// TwinCAT 3 PLC project IBF_Devices
// Title: IBF_Device
// Company: Industrial Brains B.V.
// ProjectVersion: 0.0.0.0
// ProgramVersion: 3.1.4022.4
// CompilerDefines: InclSerialCom := 'true'
// libraries:
//   IBF_Utilities, * (Industrial Brains B.V.)
//   Tc2_Math, * (Beckhoff Automation GmbH)
//   Tc2_MC2, * (Beckhoff Automation GmbH)
//   Tc2_MC2_Drive, * (Beckhoff Automation GmbH)
//   Tc2_Standard, * (Beckhoff Automation GmbH)
// project tree:
//   Actuators/Cylinder/DataTypes/ E_CylinderCmd.TcTLEO (not stored), E_ValveResetState.TcTLEO
//   Actuators/Cylinder/DataTypes/ManualControls/ UDT_ManualValveControl.TcDUT (not stored)
//   Actuators/Cylinder/Functions/ Fb_DevCylWithFbk.TcPOU, FB_DevValve.TcPOU (not stored)
//   Axis/DataTypes/ E_AxisCmd.TcTLEO (not stored), UDT_AxisData.TcDUT (not stored), UDT_AxVal.TcDUT, UDT_ManualAxisCtrl.TcDUT (not stored)
//   Axis/FunctionBlocks/Analog/ FB_DevAnalogAxis.TcPOU, ST_ManualAnalogAxisCtrl.TcDUT
//   Axis/FunctionBlocks/ServoHybrid/ FB_DevBasicACAxis.TcPOU (not stored), FB_DevHybridAc.TcPOU (not stored)
//   Axis/FunctionBlocks/Servo/ Fb_DevAxis.TcPOU
//   Axis/FunctionBlocks/TwoVelocityControl/DataTypes/ st_ManualDigitalMotorControl.TcDUT (not stored)
//   Axis/FunctionBlocks/TwoVelocityControl/ FB_DevTwoVelocityAxis.TcPOU (not stored)
//   Axis/Interface/ iTwoDirectionalMotor.TcIO, iTwoDirectionalMotorWithFast.TcIO (not stored)
//   BaseFunctions/ FB_DevBase.TcPOU, UDT_DevManualCtrl.TcDUT
//   Buttons/Functions/ FB_DevHMIButton.TcPOU (not stored), FB_DevPushbuttonLight.TcPOU (not stored), FB_DevPushButton.TcPOU (not stored)
//   CounterCards/FunctionBlocks/KL1512/ FB_DevKL1512.TcPOU (not stored)
//   CounterCards/FunctionBlocks/KL5151/ FB_DevKL5151.TcPOU (not stored)
//   CounterCards/Interfaces/ iCounter.TcIO (not stored)
//   CounterCards/ st_ManualCounterControl.TcDUT
//   DevTypes/ E_Devices.TcTLEO (not stored)
//   Encoders/FunctionBlocks/ FB_EncoderBase.TcPOU (not stored), FB_EncoderInput.TcPOU (not stored)
//   GroupHandlers/ GVL_DevManual.TcGVL (not stored)
//   GroupHandlers/ManualControlHandler/ FB_ManualController.TcPOU (not stored), UDT_DeviceID.TcDUT (not stored)
//   HardwareDiagnostics/ FB_ELModuleDiag.TcPOU (not stored)
//   Heaters/ FB_DevDoublePWM.TcPOU, FB_DevPWMGenerator.TcPOU (not stored)
//   Lights/Functions/ Fb_DevLight.TcPOU (not stored)
//   Outputs/AnalogOutputs/ FB_DevAnalogOutput.TcPOU (not stored), FB_DevAnalogOutputScaled.TcPOU
//   Outputs/DigitalOutputs/ FB_DevDigitalOutput.TcPOU (not stored)
//   Sensors/AnalogInput/FunctionBlocks/ FB_DevAnalogInput.TcPOU (not stored), FB_DevAnalogInputScaled.TcPOU, FB_DevHDAnalogInAutoCalibrate.TcPOU (not stored), FB_DevAnalogInAutoCalibrate.TcPOU (not stored), FB_DevHDAnalogInputScaled.TcPOU (not stored), FB_DevHDAnalogInput.TcPOU (not stored)
//   Sensors/DigitalSensor/FunctionBlocks/ Fb_DevDigitalInput.TcPOU (not stored), Fb_DevDigitalInputFunctions.TcPOU (not stored)
//   Sensors/FootPedals/DataTypes/ E_FootpedalPos.TcTLEO
//   Sensors/FootPedals/FunctionBlocks/ FB_EfkaEB301A_FootPedal.TcPOU (not stored)
//   Sensors/ModuleSpecific/EL3556_Loadcell/ Fb_DevEL3356_LoadCell.TcPOU (not stored)
//   Version/ Global_Version.TcGVL (not stored)

// ---- Axis/DataTypes/UDT_AxVal.TcDUT
TYPE UDT_AxVal :
STRUCT
	// ***** Velocity settings *****
		HardMax		: LREAL 	; // Hardware maximum set absolute maximum
		ManMax 		: LREAL		; // Manual maximum percentage of hardware max
		AutoMax		: LREAL		; // Automatic maximum percentage of hardware max
		HomeMax		: LREAL 	; // Homing maximum percentage of hardware max
		CmdVal		: LREAL 	; // Commanded value
		SafeVal		: LREAL		; // Command value after safety check
		PrevVal		: LREAL		; // previous command value 
		ActVal		: LREAL		; // Actual value
		ActModulo	: LREAL		; // [deg] Modulo position
		RefVal		: LREAL 	; // referance value (basic setting or home) 
END_STRUCT
END_TYPE

// ---- Axis/FunctionBlocks/Analog/ST_ManualAnalogAxisCtrl.TcDUT
TYPE ST_ManualAnalogAxisCtrl :
STRUCT
	bCmdRunCW	: BOOL ;
	bCmdRunCCW	: BOOL ;
	fCmdVelocity: LREAL ; 
	
END_STRUCT
END_TYPE

// ---- BaseFunctions/UDT_DevManualCtrl.TcDUT
TYPE UDT_DevManualCtrl :
STRUCT
END_STRUCT
END_TYPE

// ---- CounterCards/st_ManualCounterControl.TcDUT
TYPE st_ManualCounterControl :
STRUCT
	bManSetValue 	: BOOL ; // Set value from manual control
	nManValue		: UDINT; // Manual value
	nCount			: UDINT; // Counter value
END_STRUCT
END_TYPE

// ---- Actuators/Cylinder/DataTypes/E_ValveResetState.TcTLEO
{attribute 'qualified_only'}
{attribute 'strict'}
TYPE E_ValveResetState :
(
	Res_Idle 		:= 0,
	Res_Closed		:= 1,
	Res_Open		:= 2
);
END_TYPE

// ---- Sensors/FootPedals/DataTypes/E_FootpedalPos.TcTLEO
{attribute 'qualified_only'}
{attribute 'strict'}
TYPE E_FootpedalPos :
(
	eReverse2 	:= -2,
	eReverse1 	:= -1,
	eIdle		:= 0,
	eForward0	:= 1,
	eForward1	:= 2,
	eForward2	:= 3,
	eForward3	:= 4,
	eForward4	:= 5,
	eForward5	:= 6,
	eForward6	:= 7,
	eForward7	:= 8,
	eForward8	:= 9,
	eForward9	:= 10,
	eForward10	:= 11,
	eForward11	:= 12,
	eForward12	:= 13,
	eFalse			
) INT; 
END_TYPE
//  eReverse2 = '-2'
//  eReverse1 = '-1'

// ---- Axis/Interface/iTwoDirectionalMotor.TcIO
INTERFACE iTwoDirectionalMotor // Two directional motor control

METHOD CmdRunCCW : BOOL
VAR_INPUT
END_VAR
END_METHOD

METHOD CmdRunCW : BOOL
VAR_INPUT
END_VAR
END_METHOD

METHOD Init : BOOL
VAR_INPUT
	// Message location data
	nId				: UDINT ; // Identification number of object
	nParentId		: UDINT ; // Id of higher level If aplicable (0 = no parent)
END_VAR
END_METHOD

END_INTERFACE

// ---- Actuators/Cylinder/Functions/Fb_DevCylWithFbk.TcPOU
{attribute 'reflection'}
FUNCTION_BLOCK PUBLIC Fb_DevCylWithFbk EXTENDS FB_DevValve
VAR_INPUT
	bIcfFbkOpenPresent 	: BOOL := FALSE ; // Feedback for cylinder open is present 
	bIcfFbkClosedPresent: BOOL := FALSE ; // Feedback for Cylinder closed is present
	bIcfTimeChecked		: BOOL := TRUE 	; // Cylinder timing is checked = default true
	nMargin				: LREAL:= 10	; // % of tollerance in move speed 
END_VAR
VAR_OUTPUT
	// ===== Teach function =======
	bCmdCopyTimeParam 	: BOOL	:= FALSE 	;// Cylinder, Command to higher level copy toucht time to parameters
	bFeClosed			: BOOL 	:= FALSE	; // closed sensor falling edge
	bReClosed			: BOOL 	:= FALSE	; // closed sensor rising edge
	bFeOpen				: BOOL 	:= FALSE 	; // Open sensor falling edge
	bReOpen				: BOOL 	:= FALSE 	; // open sensor rising edge 
	bReOpenSlow         : BOOL  := FALSE    ; // rising edge, opening went too slow
	bReOpenFast         : BOOL  := FALSE    ; // rising edge, opening went too fast
	bReCloseSlow        : BOOL  := FALSE    ; // rising edge, closing went too slow
	bReCloseFast        : BOOL  := FALSE    ; // rising edge, closing went too fast
END_VAR
VAR	
	bFcoCalcDone	: BOOL := FALSE ; // Calculate timers done 
	
	stTimesClose	: Udt_TimerBandwith ; // Timer bandwith for cylinder close
	stTimesOpen		: Udt_TimerBandwith	; // Timer bandwitch for cylinder open 
	
	fbSensorClosed	: Fb_DevDigitalInputFunctions ; // Digital sensor function closed detection
	fbSensorOpen	: Fb_DevDigitalInputFunctions ; // Digital sensor function open detection
	
	fbTimerOpen		: TON ; // Timer for cylinder to open
	fbTimerClose 	: TON ; // Timer for cylinder to close
	fbTimerTeach	: TON ; // timer for teachin cylinder 

	rtCmdWriteParam	: R_TRIG ; // Write parameter rising edge trigger 
	// Simulation
	fbTimerSimOpen 	: TON 	; 
	fbTimerSimClose	: TON 	; 
	
	// Time Cylinder valid 
	bTriggerTimeClose	: BOOL ;
	bTriggerTimeOpen	: BOOL ;
END_VAR

// set device type
	IF eDevType = E_Devices.Undefined THEN 
		eDevType := E_Devices.Cylinder ;
	END_IF

// call base function 
	SUPER^(refFbFault := refFbFault);

// check for device init
	IF NOT bInitOk THEN
		RETURN;
	END_IF 

// ====== Check direction of movement =======
	ExecDirection();
	
// ====== Reset movement indicators =======
	bReOpenSlow  := FALSE;
	bReOpenFast  := FALSE;
	bReCloseSlow := FALSE;
	bReCloseFast := FALSE;

// ====== Check movement speed =======
	ExecTimeout();
	
// ====== Calculate timers =======
	CalcTimers();

METHOD PRIVATE CalcTimers : BOOL
VAR
END_VAR
IF stParTimeToClose.fValue = stTimesClose.Nominal AND stParTimeToOpen.fValue = stTimesOpen.Nominal AND bFcoCalcDone THEN 
	RETURN ;
ELSE
	bFcoCalcDone := FALSE ;
END_IF
 
// ====== Calculate close times ======
	stTimesClose.Nominal 	:= stParTimeToClose.fValue ;
	stTimesClose.Maximum 	:= stParTimeToClose.fValue * (1 + (nMargin / 100));
	stTimesClose.Minimal 	:= stParTimeToClose.fValue * (1 - (nMargin / 100));

// ====== Calculate open times ======
	stTimesOpen.Nominal 	:= stParTimeToOpen.fValue ;
	stTimesOpen.Maximum 	:= stParTimeToOpen.fValue * (1 + (nMargin / 100));
	stTimesOpen.Minimal 	:= stParTimeToOpen.fValue * (1 - (nMargin / 100));
	
// ====== Set feedback =======
	bFcoCalcDone := TRUE ;

// ===== send write parameters command ======	
	rtCmdWriteParam(CLK := bFcoCalcDone);
	bCmdCopyTimeParam := rtCmdWriteParam.Q	;
END_METHOD

METHOD PUBLIC CmdSimulate : BOOL
VAR_INPUT
	bFbkReverse		: BOOL := FALSE ; 
	tTimeSimOpen	: TIME := T#1S 	;
	tTimeSimClose	: TIME := T#1S 	;  
END_VAR
// Run timers when cylinder is active 
	fbTimerSimOpen	(IN := q_Open	, PT := tTimeSimOpen);
	fbTimerSimClose	(IN := q_Close	, PT := tTimeSimClose);

// set feedback sensors to simulate
	fbSensorOpen.bCmdSimulate 	:= TRUE ;
	fbSensorClosed.bCmdSimulate := TRUE ;

// set simulated feedback state 
	IF bFbkReverse THEN 
		fbSensorClosed.bSimState:= fbTimerSimOpen.Q 	;
		fbSensorOpen.bSimState	:= fbTimerSimClose.Q 	; 	
	ELSE 
		fbSensorClosed.bSimState:= fbTimerSimClose.Q 	;
		fbSensorOpen.bSimState	:= fbTimerSimOpen.Q 	; 	
	END_IF
END_METHOD

METHOD PUBLIC CmdTeach : BOOL
VAR_INPUT
END_VAR
// ====== turn off time check function until new calculation cycle =======
	bFcoCalcDone := false ;

// ====== teach cylinder from hardware inputs ======
	fbTimerTeach	(PT:= T#60S);
	fbTimerSwitchDir(PT:= T#1S); 
// ====== time cylinder cycles ======
	// ===== Start test loop =====
	IF bFco_Closed AND fbTimerSwitchDir.Q THEN
		bCmdClose 			:= FALSE;
		bCmdOpen 			:= TRUE ;
		fbTimerSwitchDir.IN	:= FALSE; 
		fbTimerTeach.IN 	:= TRUE ;
	ELSIF bFco_Open AND fbTimerSwitchDir.Q THEN
		bCmdClose 			:= TRUE ;
		bCmdOpen 			:= FALSE;
		fbTimerSwitchDir.IN	:= FALSE; 
		fbTimerTeach.IN 	:= TRUE ;
	ELSIF NOT bCmdClose AND NOT bCmdOpen THEN 
		bCmdClose 			:= TRUE ;
		bCmdOpen 			:= FALSE;
		fbTimerTeach.IN 	:= TRUE ;
	END_IF

// ====== start timing ========
	IF bCmdClose AND bFco_Closed THEN 
		IF fbTimerTeach.IN THEN
			stParTimeToClose.fValue 	:= TIME_TO_LREAL(fbTimerTeach.ET);
		END_IF
		fbTimerSwitchDir.IN := TRUE 		;
		fbTimerTeach.IN 	:= FALSE 		;
	ELSIF bCmdOpen AND bFco_Open THEN 
		IF fbTimerTeach.IN THEN
			stParTimeToOpen.fValue		:= TIME_TO_LREAL(fbTimerTeach.ET);
		END_IF
		fbTimerSwitchDir.IN := TRUE 		;
		fbTimerTeach.IN 	:= FALSE 		;
	END_IF
END_METHOD

METHOD PRIVATE ExecDirection : BOOL
VAR_INPUT
END_VAR
// ===== Check direction commands =====
 	IF q_Close AND fbSensorOpen.bReStatus AND NOT q_Open THEN
		stFault.Active			:= TRUE ;
		stFault.MessageNumber	:= E_MessageNumbers.CF_WrongDirection 	;
		stFault.Discription		:= CONCAT( sName,' Cylinder Opening instead of closing');
		stFault.FaultType		:= E_FaultTypes.CF 					;
		bErrorActive			:= TRUE 								;
	ELSIF q_Open AND fbSensorClosed.bReStatus AND NOT q_close THEN
		stFault.Active			:= TRUE ;
		stFault.MessageNumber	:= E_MessageNumbers.CF_WrongDirection 	;
		stFault.Discription		:= CONCAT( sName,' Cylinder closing instead of opening');
		stFault.FaultType		:= E_FaultTypes.CF 					;
		bErrorActive			:= TRUE 								;
	END_IF
END_METHOD

METHOD PROTECTED ExecSetFeedback : BOOL
VAR_INPUT
END_VAR
{warning disable C0371}
// ====== Call sensor Open function =======
	IF bIcfFbkClosedPresent THEN 
		fbSensorClosed(refFbFault := refFbFault);
		bFco_Closed := fbSensorClosed.bFcoInputActive ;
		bFeClosed 	:= fbSensorClosed.bFeStatus ;
		bReClosed 	:= fbSensorClosed.bReStatus ;
	ELSE 
		fbTOnClose	(IN 	:= q_Close, PT 	:= LREAL_TO_TIME(stParTimeToClose.fValue))	;
		bFco_Closed := fbTOnClose.Q ;
	END_IF

// ====== Call sensor Close function =======
	IF bIcfFbkOpenPresent THEN 
		fbSensorOpen(refFbFault := refFbFault) 	;
		bFco_open 	:= fbSensorOpen.bFcoInputActive ;
		bFeOpen		:= fbSensorOpen.bFeStatus;
		bReOpen		:= fbSensorOpen.bReStatus;
	ELSE 
		FbTOnOpen	(IN 	:= q_Open, PT 	:= LREAL_TO_TIME(stParTimeToOpen.fValue))	;
		bFco_Open := FbTOnOpen.Q ;
	END_IF

{warning restore C0371}
// ====== set outputs =======
	bReady		:= bFco_Closed OR bFco_Open ;
END_METHOD

METHOD PRIVATE ExecTimeout : BOOL
VAR_INPUT
END_VAR
VAR
	nTimePassedMs : LREAL ;
END_VAR
IF bFcoCalcDone AND bIcfTimeChecked AND bEnable THEN 
// ====== Set triggers ======
	IF q_Close  AND bFco_Open THEN 
		bTriggerTimeClose := TRUE ;
	ELSIF q_Open OR bFco_Closed  THEN 
		bTriggerTimeClose := FALSE ;
	END_IF

	IF q_Open  AND bFco_Closed THEN 
		bTriggerTimeOpen := TRUE ;
	ELSIF q_Close OR bFco_Open THEN
		bTriggerTimeOpen := FALSE ;
	END_IF
ELSE
	bTriggerTimeClose 	:= FALSE ;
	bTriggerTimeOpen	:= FALSE ;
END_IF


//======= run timers =======
	IF bIcfFbkClosedPresent THEN 
		fbTimerClose(IN := q_Close AND bEnable, PT := T#1M);
	END_IF	
	
	IF bIcfFbkOpenPresent THEN 
		fbTimerOpen	(IN := q_Open AND bEnable , PT := T#1M);
	END_IF

//====== Run timeout checks for cylinder close =======
	nTimePassedMs:= TIME_TO_LREAL(fbTimerClose.ET);
	
	IF bIcfFbkClosedPresent THEN 
		IF bTriggerTimeClose THEN 
			IF fbSensorClosed.bReStatus THEN 
				IF nTimePassedMs < stTimesClose.Minimal THEN 
					// send message to HMI 
					stFault.Active			:= TRUE 							;
					stFault.MessageNumber	:= E_MessageNumbers.CF_MoveToFast 	;
					stFault.Discription		:= CONCAT( sName, ' Cylinder closing to fast' )	;
					stFault.FaultType		:= E_FaultTypes.CF 					;
					bErrorActive			:= TRUE 							;
					bReCloseFast			:= TRUE                             ;
				END_IF
			ELSIF	nTimePassedMs > stTimesClose.Maximum  THEN
				// send message to HMI 
				stFault.Active			:= TRUE ;
				stFault.MessageNumber	:= E_MessageNumbers.CF_MoveToSlow		;
				stFault.Discription		:= CONCAT( sName,' Cylinder closing to Slow')	;
				stFault.FaultType		:= E_FaultTypes.CF 						;
				bErrorActive			:= TRUE 								;
				bReCloseSlow			:= TRUE                             	;
			END_IF
		END_IF
	END_IF	

//====== Run timeout checks for cylinder Open =======
	nTimePassedMs:= TIME_TO_REAL(fbTimerOpen.ET);

	IF bIcfFbkOpenPresent THEN 
		IF bTriggerTimeOpen THEN 
			IF fbSensorOpen.bReStatus THEN 
				IF nTimePassedMs < stTimesOpen.Minimal THEN 
					// send message to HMI 
					stFault.Active			:= TRUE ;
					stFault.MessageNumber	:= E_MessageNumbers.CF_MoveToFast 	;
					stFault.Discription		:= CONCAT( sName,' Cylinder Opening to fast')		;
					stFault.FaultType		:= E_FaultTypes.CF 					;
					bErrorActive			:= TRUE 							;
					bReOpenFast 			:= TRUE 							;
				END_IF
			ELSIF	nTimePassedMs > stTimesOpen.Maximum  THEN
				// send message to HMI 
				stFault.Active			:= TRUE ;
				stFault.MessageNumber	:= E_MessageNumbers.CF_MoveToSlow 	;
				stFault.Discription		:= CONCAT( sName,' Cylinder Opening to Slow')		;
				stFault.FaultType		:= E_FaultTypes.CF 					;
				bErrorActive			:= TRUE 							;
				bReOpenSlow 			:= TRUE 							;
			END_IF
		END_IF
	END_IF
END_METHOD

METHOD PUBLIC Init : BOOL
VAR_INPUT
	// Message location data
	nId			: UDINT ; // Identification number of object
	nParentId	: UDINT ; // Id of higher level If aplicable (0 = no parent)
	// Command state
	eResetState		: E_ValveResetState := 0		; // Cylinder reset state variable (default is idle) 
	eSafeState		: E_ValveResetState	:= 0		; // Valve safe state
END_VAR
bFcoCalcDone := FALSE;

// Enable sensor feedback
fbSensorClosed.bEmbeded := TRUE ;
fbSensorClosed.bEnable	:= TRUE ;
fbSensorClosed.Init	(	nId 		:= 0,
						nParentId 	:= nLocationId) ;

fbSensorOpen.bEmbeded := TRUE ;
fbSensorOpen.bEnable	:= TRUE ;
fbSensorOpen.Init	(	nId 		:= 1,
						nParentId 	:= nLocationId) ;

// Call feedback sensors 
ExecSetFeedback(); 

SUPER^.Init(nId, nParentId, eResetState, eSafeState);

// ===== Set device type for manual control =====
eDevType := E_Devices.Cylinder ;

bInitOk := fbSensorClosed.bInitOk 	AND bInitOk ;
bInitOk := fbSensorOpen.bInitOk		AND bInitOk ;
Init 	:= bInitOk ;
END_METHOD

END_FUNCTION_BLOCK

// ---- Axis/FunctionBlocks/Analog/FB_DevAnalogAxis.TcPOU
FUNCTION_BLOCK PUBLIC FB_DevAnalogAxis EXTENDS FB_DevBase
VAR_INPUT
	stManualCtrl 	: ST_ManualAnalogAxisCtrl ; // Manual control
END_VAR
VAR_OUTPUT
	bDriveOk		: BOOL ; // Drive is ok
	bMovingCW		: BOOL ; // Move CW output is active
	bMovingCCW		: BOOL ; // Move CCW output is active
	fActVelocity	: LREAL; // Command velocity of motor
END_VAR
VAR // internal functions 
	fbVelocity		: FB_DevAnalogOutputScaled 	;
	fbqRun			: FB_DevDigitalOutput		;
	fbqReset		: FB_DevDigitalOutput		;
	fbqReverse		: FB_DevDigitalOutput		;
	fbiEnabled		: Fb_DevDigitalInput		;
END_VAR
VAR // Internal commands
	fCmdVelocity	: LREAL;
	bCmdRunCW 		: BOOL ;
	bCmdRunCCW		: BOOL ;
	bCmdReset		: BOOL ;	 
	bInternalEnable : BOOL ;
END_VAR

SUPER^(refFbFault := refFbFault);

// ===== Check inputs =====
	fbiEnabled( bEmbeded	:= TRUE,
				refFbFault 	:= refFbFault);

IF bInitOk THEN 
	ExecSetOutputs() ;
	bDriveOk	:= fbiEnabled.bFcoInputActive ;
END_IF

METHOD PUBLIC CmdManual : BOOL
VAR_INPUT
END_VAR
bCmdManual := TRUE ;

// Execute Manual commands
	IF stManualCtrl.bCmdRunCW THEN 
		CmdRunCW(fCmdVelocity := stManualCtrl.fCmdVelocity);
	ELSIF stManualCtrl.bCmdRunCCW THEN 
		CmdRunCCW(fCmdVelocity := stManualCtrl.fCmdVelocity);
	END_IF
END_METHOD

METHOD PUBLIC CmdReset : BOOL
VAR_INPUT
END_VAR
bErrorActive 	:= FALSE;

bCmdReset		:= TRUE ;

CmdReset		:= TRUE ;
END_METHOD

METHOD PUBLIC CmdRunCCW : BOOL
VAR_INPUT
	fCmdVelocity	: LREAL ; // Command velocity
END_VAR
bCmdRunCCW			:= TRUE ;
THIS^.fCmdVelocity 	:= fCmdVelocity ; 

CmdRunCCW 	:= bMovingCW ;
END_METHOD

METHOD PUBLIC CmdRunCW : BOOL
VAR_INPUT
	fCmdVelocity	: LREAL ; // Command velocity
END_VAR
bCmdRunCW := TRUE ;
THIS^.fCmdVelocity 	:= fCmdVelocity ;

CmdRunCW 	:= bMovingCW ;
END_METHOD

METHOD PUBLIC CmdSafeStop : BOOL
VAR_INPUT
END_VAR
bIsSafe := TRUE ;

bIsSafe := fbVelocity.CmdSafeStop() AND bIsSafe ;
bIsSafe := fbqRun.CmdSafeStop() 	AND bIsSafe ;
bIsSafe := fbqReverse.CmdSafeStop() AND bIsSafe ;
bIsSafe := fbqReset.CmdSafeStop() 	AND bIsSafe ;

CmdSafeStop := bIsSafe;
END_METHOD

METHOD PRIVATE ExecSetOutputs : BOOL
VAR_INPUT
END_VAR
// ====== Check safety and enable ======
IF bSafetyOk 
AND fbiEnabled.bFcoInputActive 
AND (bEnable OR bManual) THEN 
	bInternalEnable := TRUE;
ELSE
	fCmdVelocity 	:= 0;
	bCmdRunCW		:= FALSE;
	bCmdRunCCW		:= FALSE;
END_IF 

{warning disable C0371}
// ====== Set outputs =======
	fbVelocity	(	bEmbeded 	:= TRUE,
					bSafetyOk	:= bSafetyOk,
					bEnable		:= bInternalEnable,
					fCmdValue	:= fCmdVelocity, 
					refFbFault	:= refFbFault);
				
	fbqRun		(	bEmbeded 	:= TRUE,
					bSafetyOk	:= bSafetyOk,
					bEnable		:= bInternalEnable,
					bCmdOn		:= bCmdRunCW OR bCmdRunCCW,
					refFbFault	:= refFbFault);
				
	fbqReverse	(	bEmbeded 	:= TRUE,
					bSafetyOk	:= bSafetyOk,
					bEnable		:= bInternalEnable,
					bCmdOn		:= bCmdRunCCW,
					refFbFault	:= refFbFault);

	fbqReset	(	bEmbeded 	:= TRUE,
					bSafetyOk	:= bSafetyOk,
					bEnable		:= bInternalEnable,
					bCmdOn		:= bCmdReset,
					refFbFault	:= refFbFault);
{warning restore C0371}
// ===== reset input commands =====
	fCmdVelocity 	:= 0;
	bCmdRunCW		:= FALSE;
	bCmdRunCCW		:= FALSE;
	bCmdManual		:= FALSE;
	bCmdReset		:= FALSE;
	bInternalEnable := FALSE;
// ===== set feedback =====

bMovingCW		:= fbqRun.bOutputState AND NOT fbqReverse.bOutputState;
bMovingCCW		:= fbqRun.bOutputState AND fbqReverse.bOutputState;
fActVelocity	:= fbVelocity.fOutputValue ;
END_METHOD

METHOD Init : BOOL
VAR_INPUT
	// Message location data
	nId			: UDINT ; // Identification number of object
	nParentId	: UDINT ; // Id of higher level If aplicable (0 = no parent)

	// Motor settings
	fMaxVelocity : LREAL ; // Maximum motor velocity for scaling
END_VAR
// ====== initialize components =====
	bInitOk := TRUE ;

// ====== Calculate device id =====
	bInitOk :=	ExecIdentifyDevice(nId,nParentId, E_ComponentTypes.Axis) AND bInitOk;

// ====== Set manual device type ======
	eDevType := E_Devices.AnalogAxis ;	


bInitOk := 	fbVelocity.Init	( 	nId 			:= 0,
								nParentId		:= nLocationId,
								benableNegative	:= FALSE )
								AND bInitOk;
			fbVelocity.SetScaling	(fMaxValue 		:= fMaxVelocity);
								
bInitOk	:= 	fbqRun.Init		( 	nId				:= 1,
								nParentId		:= nLocationId)
								AND bInitOk;

bInitOk	:= 	fbqReset.Init	( 	nId				:= 2,
								nParentId		:= nLocationId)
								AND bInitOk;

bInitOk	:= 	fbqReverse.Init	( 	nId				:= 3,
								nParentId		:= nLocationId)
								AND bInitOk;

bInitOk	:= 	fbiEnabled.Init	( 	nId				:= 4,
								nParentId		:= nLocationId)
								AND bInitOk;

// ====== Set feedback =======
Init := bInitOk;
END_METHOD

END_FUNCTION_BLOCK

// ---- BaseFunctions/FB_DevBase.TcPOU
{attribute 'reflection'}
FUNCTION_BLOCK PUBLIC FB_DevBase EXTENDS FB_FunctionBase
VAR_INPUT
	bEmbeded		: BOOL 	:= FALSE ; // Device is embedded into another device (not added to manual screen)
	// function references 
	refFbManualCtrl	: REFERENCE TO FB_ManualController := GVL_DevManual.fbManualControler; // reference to manual handler
END_VAR
VAR_OUTPUT
	eDevType		: E_Devices		:= E_Devices.Undefined	; // Type of Device 	
END_VAR
VAR
	// Manual control variables
	bAddedToManual	: BOOL 	:= FALSE 	; // device is added tot manual control function 	
END_VAR

SUPER^(refFbFault := refFbFault);

// Add device to manual screen
IF NOT bEmbeded THEN 
	IF bInitOk
	AND NOT bAddedToManual 
	AND sName <> '' 
	AND __ISVALIDREF(refFbManualCtrl)
	THEN 
		bAddedToManual S= refFbManualCtrl.CmdAddDevice(THIS^);
	END_IF
END_IF

METHOD PUBLIC CmdManual : BOOL
VAR_INPUT
END_VAR
bCmdManual := true ;
END_METHOD

METHOD PUBLIC CmdSafeStop : BOOL
VAR_INPUT
END_VAR
// check if device is safe
bIsSafe 	:= NOT bSafetyOk ;
CmdSafeStop := bIsSafe ;
END_METHOD

END_FUNCTION_BLOCK

// ---- Outputs/AnalogOutputs/FB_DevAnalogOutputScaled.TcPOU
{attribute 'reflection'}
FUNCTION_BLOCK FB_DevAnalogOutputScaled EXTENDS FB_DevAnalogOutput
VAR_INPUT
END_VAR
VAR_OUTPUT
END_VAR
VAR
	fGainFactor 	: LREAL:= 32767	;
END_VAR

SUPER^(refFbFault := refFbFault);

METHOD INTERNAL ExecSetFeedback : BOOL
VAR_INPUT
END_VAR
// Set feedback 
fOutputValue := qnHwOut ;
END_METHOD

METHOD INTERNAL ExecSetOutput : BOOL
VAR_INPUT
END_VAR
// Set Output to physical device
IF bSafetyOk AND (bEnable OR bCmdManual) THEN 
	qnHwOut := LREAL_TO_INT(fCmdValue * fGainFactor) ;
	qnHwOut := LIMIT(nLimitMin, qnHwOut, nLimitMax) ; 
ELSE 
	qnHwOut		:= 0;
	fCmdValue 	:= 0 ; 
END_IF
END_METHOD

METHOD PUBLIC SetScaling : BOOL 
VAR_INPUT
	fMaxValue	: LREAL ; 		// Maximum input value after scaling, e.g. 100% (mandatory input)  
END_VAR
// calculate gain 
fGainFactor := nLimitMax / fMaxValue ;
END_METHOD

END_FUNCTION_BLOCK

// ---- Axis/FunctionBlocks/Servo/Fb_DevAxis.TcPOU
{attribute 'reflection'}
FUNCTION_BLOCK PUBLIC Fb_DevAxis EXTENDS FB_DevBase
VAR_INPUT
	// ===== General Function input =====
		fCmdAcc			: LREAL := 15000;
		fCmdDecc		: LREAL := 15000; 
	// ===== Master Axis =====
		refMasterAxis	: REFERENCE TO AXIS_REF ; // Master axis reference (if applicable)
		bReverseSlave	: BOOL 	:= FALSE; // Reverse slave axis relative to master
		fCmdGearRatio	: LREAL := 1 ; // Gear ratio Master/Slave (1/Ratio) 
	// Manual control reference
		stManualCtrl	: UDT_ManualAxisCtrl ;
END_VAR
VAR_OUTPUT
	// ====== State indications =======
		bHomed			: BOOL 	:= FALSE; 
		bError 			: BOOL 	:= FALSE;
		bStopped		: BOOL 	:= FALSE;
		bResetDone		: BOOL 	:= FALSE;
		bGearedAsSlave	: BOOL 	:= FALSE;
		bVelocityLimited: BOOL 	:= FALSE;  
		bIdle			: BOOL 	:= FALSE;
		fVelocity		: LREAL	:= 0	; // Axis velocity [rpm or units/sec] depending on config
		fActPosition	: LREAL := 0	; // Axis actual position [Units] depending on config	
		bReInTargetPos	: BOOL 	:= false; // rising edge axis is in position
	// ====== axis reference ======
		AxisRef			: AXIS_REF	; // Axis reference to hardware 
	// ====== Axis Settings ======
		fMaxVelo		: LREAL := 0 ; // Axis Maximum velocity
		fMaxAcc			: LREAL := 0 ; // Axis Maximum cceleration
		fMaxDec			: LREAL := 0 ; // axis Maxium deceleration 
	
//		fSafeVeloLimit	: LREAL	:= 200; // Safe velocity limit 
		tEnableDelay	: TIME 	:= T#0MS	;
		tDisableDelay	: TIME 	:= T#500MS  ;
	// ==== Axis data ====
		fEncoderTurnoverValue	: LREAL ;   
		
END_VAR
VAR // Axis configuration 
	// ===== HW Config Bits =====
		bIcfCmdVelocityRpm	: BOOL ; // input speeds in Rpm
		bIcfEnableForward 	: BOOL ; // Enable forward motion
 		bIcfEnablereverse	: BOOL ; // Enable reverse motion
		bIcfAlwaysEnable	: BOOL ; // 1 = Axis always enabled, 0 = Axis disabled at Idle 
		bIcfSimulationMode	: BOOL := FALSE ; // Simulation mode is active [default set to False] 
		bIcfModuloAxis		: BOOL := FALSE ; // Show axis position as modulo
		bIcfSTOPresent		: BOOL := FALSE ; // Axis Safe torque off is present
		bIcfNCHomeSensor	: BOOL := FALSE ; // Homing sensor is inverted (NC)	
	// ===== Internal motion values ======
		fHomePosition		: LREAL := 0 ; // set position at homing
	// Command Modes
		mcHomingMode 		: MC_HomingMode := MC_direct ; // Homing Mode ( MC_DefaultHoming, MC_Direct, MC_ForceCallibration, MC_ResetCallibration)
	// Values from system
		McReadSysVelo		: MC_ReadParameter		; // Read Acceleration parameter from drive 
		McReadSysAcc		: MC_ReadParameter		; // Read Acceleration parameter from drive 
		McReadSysDec		: MC_ReadParameter		; // Read Acceleration parameter from drive 
END_VAR
VAR	// ====== Axis enable =====
		bCmdEnableAxis 		: BOOL 	:= FALSE; // Command to enable the axis (External)
		bInternalEnable		: BOOL 	:= FALSE; // internal enable command (turns off after set time, and on at new motion command
		bAxisIsEnabled		: BOOL 	:= false; // Axis is enabled and ready for commands
		bDelayedEnable		: BOOL 	:= false; // Delayed enable signal for motion commands
		TonMotionEnable		: TON 			; // Timer on for motion command enable
		TofIntAxisEnable	: TOF  			; // Timer off for internal axis enable 
		bSTOOK				: BOOL 	:= FALSE; // Axis safet torque off is ok
		tonSTOOK			: TON	; // Safe torque off ok timer
	// Parameter read status 
		Cmd_EnDriveParRead	: BOOL 			; // Enable parameter read 
	// ===== Physical Homing signal =====
		IAxisHome 	AT %I* 	: BOOL 			; // Axis homing sensor from PLC (if MC_DefaultHoming is used)
		IAxisSTOOK	AT %I* 	: BOOL 			; // Axis STO is ok
END_VAR
VAR	// =============== Motion status functions ================
	// =============== Motion function blocks =================
		fbMcPower 			: MC_Power		;		// FB for enable and override
		fbMcReset 			: MC_Reset		;		// FB to reset axis
		fbSoeReset			: FB_SoEReset	; 		// FB to reset axis hardware
		fbMcHome			: MC_Home		;		// Fb to home Axis
		fbMcStop 			: MC_Stop		;		// FB to stop axis
		fbMcHalt			: MC_Halt		;		// FB to halt axis
		fbMcJog				: MC_Jog		;		// FB to Jog axis
		fbMcMoveVelocity	: MC_MoveVelocity;		// FB to move with specified velocity until Next command is given
		fbMcGearInSlave		: MC_GearIn		;		// FB to gear axis to master 
		fbMcGearInDyn		: MC_GearInDyn	;		// FB to gear axis dynamicly to master
		fbMcGearOutSlave	: MC_GearOut	;		// FB to decouple gearing
		fbMcSetPosition		: MC_SetPosition;		// FB to Set axis position
//		fbMcWriteParameter	: MC_WriteParameterPersistent ; // FB to write parameters in persistend data

	(* PtoP Motion move commands are in arrays so multiple commands can be stacked *) 
		fbMCMoveRelative	: ARRAY [0..1] OF MC_MoveRelative	;		// FB to move relative
		fbMcMoveAbsolute	: ARRAY [0..1] OF MC_MoveAbsolute	;		// FB to move axis (velocity movement)
		fbMcMoveModulo		: ARRAY [0..1] OF MC_MoveModulo		;		// FB to move axis to modulo position
	// ===== Safe commands =====
		bCmdSafeStop		: BOOL ;
		bCmdSafeSpeed		: BOOL ; 
	// ===== Function execute triggers =====
		bExec_Reset					: BOOL := FALSE; // Execute reset
		bExec_Halt					: BOOL := FALSE; // Execute hold
		bExec_Home					: BOOL := FALSE; // Execute Home
		bExec_JogPositive			: BOOL := FALSE; // Execute Jog in positive direction
		bExec_JogNegative			: BOOL := FALSE; // Execute Jog in negative direction
		bExec_MoveVelocity			: BOOL := FALSE; // Execute move velocity
		bExec_MoveVelocityDynamic	: BOOL := FALSE; // Execute move velocity
		bExec_GearAsSlave			: BOOL := FALSE; // Execute gear as slave
		bExec_GearSlaveDyn			: BOOL := FALSE; // Execute gear slave dynamic
		bExec_GearOutSlave			: BOOL := FALSE; // Execute gear out slave
		bExec_SetPosition			: BOOL := FALSE; // execute set position
		
	(* PtoP Motion move commands are in arrays so multiple commands can be stacked *) 
		arExec_MoveRelative	: ARRAY [0..1] OF BOOL ; // Execute move relative
		arExec_MoveAbs		: ARRAY [0..1] OF BOOL ; // Execute move absolute reverse
		arExec_MoveModulo	: ARRAY [0..1] OF BOOL ; // Execute move modulo

		tonResetDone		: TON := (PT := T#300MS) ;

	// ===== Move ristrictions ======
		bCmdLimitVelocity 	: BOOL := FALSE			; // velocity limiting is active 
		bCmdManualAccDec	: BOOL := FALSE			; // Activate manual aceleration and deceleration settings
		fCmdVelocityLimit	: LREAL:= 100			; // Maximum velocity limit when velocity limiting is active  
		fSafeOverride		: LREAL:= 10 			; // [%] Safe velocity override  
		
	// ===== Internal variables =======
		fAcceleration		: LREAL := 0 ; // Acceleration used for functions 
		fDeceleration		: LREAL := 0 ; // Deceleration used for functions
END_VAR
VAR
	// ===== Loop variables =====
		i : DINT := 0 ; // For loop increment
	// ===== check variable ======
		rtrigInPosition	: R_TRIG ; // in position trigger
	// ===== Par write timer ===== 
END_VAR
VAR // Parameters 
	ParAccManualScaling	: Udt_Parameter := (fValue := 50, fFactory := 50, bTeachable := FALSE)  ; // Acceleration scaling factor for manual functions 
	ParDecManualScaling	: Udt_Parameter := (fValue := 50, fFactory := 50, bTeachable := FALSE)	; // Deceleration scaling factor for manual functions 
END_VAR

// Call base function
SUPER^(refFbFault := refFbFault);

// ==== Check if axis is initiated =====
IF NOT bInitOk THEN 
	RETURN ; 
END_IF
// ===== Execute safe functions =====
	ExecSafeFunctions(); 
	
// ==== Execute organizational functions =====
	CallOrganizationFunctions();
// ==== execute motion functions =====
	CallMotionFunctions();

METHOD PRIVATE CallMotionFunctions : BOOL
VAR_INPUT
END_VAR
// ===== Set acceleratio and deceleration values =======
	IF bCmdManualAccDec THEN 
		fAcceleration 		:= fCmdAcc * (ParAccManualScaling.fvalue / 100);
		fDeceleration		:= fCmdDecc* (ParDecManualScaling.fValue / 100);
		bCmdManualAccDec 	:= FALSE;
	END_IF

// ===== block all other commands if axis is coupled =====
	IF NOT AxisRef.Status.Coupled THEN 
	// ===== Homing functions =====
		ExecHome		(); 
	
	// ===== Motion standstil commands =====
		ExecHalt		();
	
	// ===== Motion move functions
		ExecJog			();
		ExecMoveAbsolute();
		ExecMoveRelative();
		ExecMoveModulo	();
		ExecMoveVelocity();
	END_IF
	
// ===== Execute gearing functions =====
 IF __ISVALIDREF (refMasterAxis) THEN 
	ExecGearOut		();
	ExecGearIn		();
	ExecGearDynamic	();
 END_IF
	
// ====== reset velocity lmiting =====
	bVelocityLimited	:= bCmdLimitVelocity ;	
	bCmdLimitVelocity 	:= FALSE ; 

// ====== Reset acceleration deceleration values ======
	fAcceleration	:= fCmdAcc;
	fDeceleration	:= fCmdDecc;
END_METHOD

METHOD PRIVATE CallOrganizationFunctions : BOOL
VAR_INPUT
END_VAR
// ==== execute organizational functions =====
	ExecReadStatus		(); 
	ExecEnable			();
	ExecReset			();
//	ExecWriteParameter	();
	ExecSetPosition		();
END_METHOD

METHOD PUBLIC CmdGearDynamic : BOOL // Set axis to geared, activates with variable gear ratio until geared out or stopped (if method is no longer called then gear ratio is locked to last value)
VAR_INPUT
	fGearRatio	:	LREAL	:= 1	; // Slave Axis gearing ratio (Master = 1/ fGearRatio = Slave)	
END_VAR
// check if master is present
	IF NOT __ISVALIDREF (refMasterAxis) THEN 
		bError					:= TRUE							;
		stFault.Active 			:= TRUE 						;
		stFault.MessageNumber	:= E_MessageNumbers.FF_AxisFault;
		stFault.Discription		:= CONCAT('Axis master not found ', UDINT_TO_STRING(fbMcHalt.ErrorID));
		stFault.Discription		:= CONCAT( sName , stfault.Discription ) ;
		stFault.FaultType		:= E_FaultTypes.FF				;
	END_IF


// set blocked command if halt is active 
	bBlockedCommand 		:= fbMcHalt.Active ;


// check if command buffer is empty 
	IF AxisRef.Status.CmdBuffered THEN 
		RETURN ;
	END_IF 

// Set command to true 
	bExec_GearSlaveDyn 	:= TRUE ;
	bInternalEnable		:= TRUE ;

// coppy parameters
	fCmdGearRatio 		:= fGearRatio ;

// Set feedback output 
	CmdGearDynamic 		:= bGearedAsSlave ;
END_METHOD

METHOD PUBLIC CmdGearIn : BOOL // Set axis to geared, activates with constant gear ratio until geared out or stopped
VAR_INPUT
	fGearRatio	:	LREAL	:= 1	; // Slave Axis gearing ratio (Master = 1/ fGearRatio = Slave)	
END_VAR
// Check if master is present
	IF NOT __ISVALIDREF (refMasterAxis) THEN 
		bError					:= TRUE							;
		stFault.Active 			:= TRUE 						;
		stFault.MessageNumber	:= E_MessageNumbers.FF_AxisFault;
		stFault.Discription		:= CONCAT('Axis master not found ', UDINT_TO_STRING(fbMcHalt.ErrorID));
		stFault.Discription		:= CONCAT( sName , stfault.Discription ) ;
		stFault.FaultType		:= E_FaultTypes.FF				;
	END_IF

// set blocked command if halt is active 
	bBlockedCommand := fbMcHalt.Active ;

// check if command buffer is empty 
	IF AxisRef.Status.CmdBuffered THEN 
		RETURN ;
	END_IF 
	
// Set command to true 
	bExec_GearAsSlave 	:= TRUE ;
	bInternalEnable		:= TRUE ;

// coppy parameters
	fCmdGearRatio 				:= fGearRatio ;

// Set feedback output 
	CmdGearIn := bGearedAsSlave ;
END_METHOD

METHOD CmdGearOut : BOOL
VAR_INPUT
END_VAR
// Check if master is present
	IF NOT __ISVALIDREF (refMasterAxis) THEN 
		bError					:= TRUE							;
		stFault.Active 			:= TRUE 						;
		stFault.MessageNumber	:= E_MessageNumbers.FF_AxisFault;
		stFault.Discription		:= CONCAT('Axis master not found ', UDINT_TO_STRING(fbMcHalt.ErrorID));
		stFault.Discription		:= CONCAT( sName , stfault.Discription ) ;
		stFault.FaultType		:= E_FaultTypes.FF				;
	END_IF

// set blocked command if halt is active 
bBlockedCommand := fbMcHalt.Active ;

// Set command to true
bExec_GearOutSlave 	:= TRUE ;
bExec_GearAsSlave	:= FALSE;
bExec_GearSlaveDyn 	:= FALSE;

// Set feedback Output
CmdGearOut := fbMcGearOutSlave.Done;
END_METHOD

METHOD PUBLIC CmdHalt : BOOL
VAR_INPUT
	fDeceleration 	: LREAL := 0 ; // command deceleration
	mcBuffermode	: MC_BufferMode ; // Buffermode defines how the previous command is executed.
END_VAR
// Set command to true 
bExec_Halt 		:= TRUE ;
bInternalEnable	:= TRUE ;

// coppy parameters
fbMcHalt.Deceleration	:= fDeceleration;
fbMcHalt.BufferMode		:= mcBuffermode	;

// Set feedback output 
CmdHalt := fbMchalt.Active OR fbMcHalt.Done ;
END_METHOD

METHOD PUBLIC CmdHold : BOOL
VAR_INPUT
END_VAR
// Set command to true 
bExec_Halt 		:= TRUE ;
bInternalEnable	:= TRUE ;

// coppy parameters
fbMcHalt.Deceleration	:= 0;
fbMcHalt.BufferMode		:= 0;

// Set feedback output 
CmdHold := fbMchalt.Active OR fbMcHalt.Done ;
END_METHOD

METHOD PUBLIC CmdHome : BOOL // start axis homing procedure
VAR_INPUT
	fPosition 		: LREAL := 0 ; // Homing position
END_VAR
// set blocked command if halt is active 
bBlockedCommand := fbMcHalt.Active ;

// set command to true 
bExec_Home 		:= TRUE	; 
bInternalEnable	:= TRUE ;

// coppy parameters
fbMcHome.Position 	:= fPosition 	;

// Set feedback output
CmdHome := fbMcHome.Done ;
END_METHOD

METHOD PUBLIC CmdJog : BOOL // Jog axis with variable speed. jog stops as soon as the command is false
VAR_INPUT
	fVelocity		: LREAL 	; // jog velocity can be adjusted as long as the command is active
	fPos			: LREAL 	; // Jog position or step size (if aplicable)
	bJogNegative 	: BOOL 		:= FALSE ; // jog in negative direction
	eJogmode		: E_JogMode := E_JogMode.MC_JOGMODE_CONTINOUS ; // jogmode [default MC_JOGMODE_CONTINOUS] 
END_VAR
// set blocked command if halt is active 
bBlockedCommand := fbMcHalt.Active ;

// Velocity conversion from RPM to deg/sec
	IF bIcfCmdVelocityRpm THEN 
		fVelocity := Rpm_To_DegS(fVelocity);
	END_IF

// Set command to true
	IF fbMcJog.Velocity = fVelocity THEN // If command velocity changes, then set exec to false for one cycle to trigger new velocity so the jog follows the set velocity
		bExec_JogPositive	:= NOT bJogNegative ;
		bExec_JogNegative 	:= bJogNegative ;
	END_IF
	bInternalEnable			:= TRUE ;

// coppy parameters
	fbMcJog.Velocity	:= fVelocity 	;
	fbmcjog.Mode		:= eJogmode		;
	fbMcJog.Position	:= fPos			;

// Set feedback output 
	CmdJog := fbMcJog.Active ;
END_METHOD

METHOD PUBLIC CmdKeepEnabled : BOOL
VAR_INPUT
END_VAR
// Keep internal enable on while command is active
bInternalEnable			:= TRUE ;
END_METHOD

METHOD PUBLIC CmdLimitVelocity : BOOL // limit axis maximum velocity, stays active as long as command is called. 
VAR_INPUT
	fVelocityLimit	: LREAL ; // velocity Maximum limit
END_VAR
// set blocked command if halt is active 
bBlockedCommand := fbMcHalt.Active ;

// Set velocity limiting command 
bCmdLimitVelocity S= TRUE;
	
// Set velocity maximum value 
fCmdVelocityLimit := fVelocityLimit ; 

// set feedback 
CmdLimitVelocity := bVelocityLimited ;
END_METHOD

METHOD PUBLIC CmdManual : BOOL
VAR
	eJogmode		: E_JogMode := E_JogMode.MC_JOGMODE_CONTINOUS ; // jogging mode 
END_VAR
// set blocked command if halt is active 
bBlockedCommand := fbMcHalt.Active ;

// Enable axis for manual control
bCmdManual := TRUE ;

// check safety 
IF NOT bSafetyOk THEN 
	RETURN;
END_IF

// set jog mode 
IF stManualCtrl.bCmdInching THEN 
	eJogmode := E_JogMode.MC_JOGMODE_INCHING ;
END_IF

// execute motion commands
IF stManualCtrl.bCmdJogForward OR stManualCtrl.bCmdJogReverse THEN 
	CmdJog (fVelocity := stManualCtrl.fVelocity, 
			fPos := stManualCtrl.fDistance, 
			bJogNegative := stManualCtrl.bCmdJogReverse, 
			eJogmode := eJogmode);
ELSIF stManualCtrl.bCmdToPos THEN 
	CmdMoveAbs( fPosition := stManualCtrl.fPosition, 
				fVelocity := stManualCtrl.fVelocity, 
				mcBuffermode := MC_BufferMode.MC_Aborting);
ELSIF stManualCtrl.bCmdHome THEN 
	CmdHome( fPosition := 0);
ELSE 
	CmdHalt( 	fDeceleration := fMaxDec * 0.9, 
				mcBuffermode := MC_BufferMode.MC_Aborting) ; 
END_IF
END_METHOD

METHOD PUBLIC CmdManualAccDec : BOOL
VAR_INPUT
END_VAR
bCmdManualAccDec := TRUE;

CmdManualAccDec := TRUE;
END_METHOD

METHOD PUBLIC CmdMoveAbs : BOOL // Move absolute command
VAR_INPUT
	fPosition	:	LREAL 	; // target position
	fVelocity	: 	LREAL 	; // Maximum velocity [units/sec]
	mcBuffermode: 	MC_BufferMode ; // Buffermode defines how the previous command is executed.
END_VAR
// set blocked command if halt is active 
bBlockedCommand := fbMcHalt.Active ;

// Velocity conversion from RPM to deg/sec
	IF bIcfCmdVelocityRpm THEN 
		fVelocity := Rpm_To_DegS(fVelocity);
	END_IF

// Determine function for command stacking
IF NOT AxisRef.Status.CmdBuffered OR mcBuffermode <> MC_Aborting THEN 
	IF fbMcMoveAbsolute[0].Active THEN 
		arExec_MoveAbs[1] 				:= (fPosition <> fbMcMoveAbsolute[0].Position OR fVelocity <> fbMcMoveAbsolute[0].Velocity) ;
		fbMcMoveAbsolute[1].Position 	:= fPosition ;
		fbMcMoveAbsolute[1].Velocity 	:= fVelocity ; 
		fbMcMoveAbsolute[1].BufferMode 	:= mcBuffermode ;
	ELSE
		arExec_MoveAbs[0] 				:= (fPosition <> fbMcMoveAbsolute[1].Position OR fVelocity <> fbMcMoveAbsolute[1].Velocity) ;
		fbMcMoveAbsolute[0].Position 	:= fPosition ;
		fbMcMoveAbsolute[0].Velocity 	:= fVelocity ; 
		fbMcMoveAbsolute[0].BufferMode 	:= mcBuffermode ;
	END_IF
END_IF
	
bInternalEnable	:= TRUE ;

// set feedback
IF arExec_MoveAbs[1] OR fbMcMoveAbsolute[1].Busy THEN 
	CmdMoveAbs :=	fbMcMoveAbsolute[1].Active ;
ELSE 
	CmdMoveAbs :=	fbMcMoveAbsolute[0].Active ;
END_IF
END_METHOD

METHOD PUBLIC CmdMoveModulo : BOOL // Move to a modulo position
VAR_INPUT
	fPosition	:	LREAL 	; // target position
	fVelocity	: 	LREAL 	; // Maximum velocity [units/sec]
	mcDirection : 	MC_Direction := MC_Direction.MC_Positive_Direction ; // Direction of movement mc_direction [ deafult mc_positive_direction]
	mcBuffermode: 	MC_BufferMode ; // Buffermode defines how the previous command is executed.
END_VAR
// set blocked command if halt is active 
bBlockedCommand := fbMcHalt.Active ;


// Velocity conversion from RPM to deg/sec
	IF bIcfCmdVelocityRpm THEN 
		fVelocity := Rpm_To_DegS(fVelocity);
	END_IF

// Determine function for command stacking
IF NOT AxisRef.Status.CmdBuffered OR mcBuffermode <> MC_Aborting THEN 
	IF fbMcMoveModulo[0].Busy THEN 
		arExec_MoveModulo[1] 		:= (fPosition <> fbMcMoveModulo[0].Position OR fVelocity <> fbMcMoveModulo[0].Velocity)	;
		fbMcMoveModulo[1].Velocity 	:= fVelocity 	;
		fbMcMoveModulo[1].Position 	:= fPosition 	;
		fbMcMoveModulo[1].Direction	:= mcDirection	;
		fbMcMoveModulo[1].BufferMode:= mcBuffermode ;
	ELSE    
		arExec_MoveModulo[0] 		:= (fPosition <> fbMcMoveModulo[1].Position OR fVelocity <> fbMcMoveModulo[1].Velocity) ;
		fbMcMoveModulo[0].Velocity 	:= fVelocity 	;
		fbMcMoveModulo[0].Position 	:= fPosition 	;
		fbMcMoveModulo[0].Direction	:= mcDirection	;
		fbMcMoveModulo[0].BufferMode:= mcBuffermode ;
	END_IF
END_IF 
	
bInternalEnable	:= TRUE ;

// set feedback
IF arExec_MoveModulo[1] OR fbMcMoveModulo[1].Busy THEN 
	CmdMoveModulo :=	fbMcMoveModulo[1].Active OR fbMcMoveModulo[1].Done;
ELSE
	CmdMoveModulo :=	fbMcMoveModulo[0].Active OR fbMcMoveModulo[0].Done ;
END_IF
END_METHOD

METHOD CmdMoveRelative : BOOL // move relative command 
VAR_INPUT
	fDistance	:	LREAL 	; // target position
	fVelocity	: 	LREAL 	; // Maximum velocity [units/sec]
	mcBuffermode: 	MC_BufferMode ; // Buffermode defines how the previous command is executed.
END_VAR
// set blocked command if halt is active 
bBlockedCommand := fbMcHalt.Active ;

// Velocity conversion from RPM to deg/sec
	IF bIcfCmdVelocityRpm THEN 
		fVelocity := Rpm_To_DegS(fVelocity);
	END_IF

// Determine function for command stacking
IF NOT AxisRef.Status.CmdBuffered OR mcBuffermode <> MC_Aborting THEN 
	IF fbMCMoveRelative[0].Active THEN 
		arExec_MoveRelative[1] := (fDistance <> fbMCMoveRelative[0].Distance OR fVelocity <> fbMCMoveRelative[0].Velocity) ;
		fbMCMoveRelative[1].Velocity	:= fVelocity 	;
		fbMCMoveRelative[1].Distance	:= fDistance	;
		fbMCMoveRelative[1].BufferMode	:= mcBuffermode	;
	ELSE 
		arExec_MoveRelative[0] := (fDistance <> fbMCMoveRelative[1].Distance OR fVelocity <> fbMCMoveRelative[1].Velocity) ;
		fbMCMoveRelative[0].Velocity	:= fVelocity 	;
		fbMCMoveRelative[0].Distance	:= fDistance	;
		fbMCMoveRelative[0].BufferMode	:= mcBuffermode	;
	END_IF
END_IF
bInternalEnable	:= TRUE ;

// set feedback
IF arExec_MoveRelative[1] OR fbMCMoveRelative[1].Busy THEN 
	CmdMoveRelative :=	fbMCMoveRelative[1].Active ;
ELSE
	CmdMoveRelative :=	fbMCMoveRelative[0].Active ;
END_IF
END_METHOD

METHOD PUBLIC CmdMoveVelocity : BOOL // Move with set velocity until stopped
VAR_INPUT
	fVelocity	: 	LREAL 	; // Maximum velocity [units/sec]
	mcDirection : 	MC_Direction := MC_Direction.MC_Positive_Direction ; // Direction of movement mc_direction [ deafult mc_positive_direction]
	mcBuffermode: 	MC_BufferMode ; // Buffermode defines how the previous command is executed.
END_VAR
// set blocked command if halt is active 
bBlockedCommand := fbMcHalt.Active ;

// Velocity conversion from RPM to deg/sec
	IF bIcfCmdVelocityRpm THEN 
		fVelocity := Rpm_To_DegS(fVelocity);
	END_IF

// Set command to true 
	IF NOT AxisRef.Status.CmdBuffered OR mcBuffermode <> MC_Aborting THEN 
		bExec_MoveVelocity 	:= TRUE ;
		bInternalEnable		:= TRUE ;
	END_IF
	
// coppy parameters
	fbMcMoveVelocity.Velocity	:= fVelocity 	;
	fbMcMoveVelocity.Direction 	:= mcDirection	;
	fbMcMoveVelocity.BufferMode	:= mcBuffermode	;

// Set feedback output 
	CmdMoveVelocity := fbMcMoveVelocity.Active ;
END_METHOD

METHOD PUBLIC CmdMoveVelocityDynamic : BOOL // Move with set velocity until stopped
VAR_INPUT
	fVelocity	: 	LREAL 	; // Maximum velocity [units/sec]
	mcDirection : 	MC_Direction := MC_Direction.MC_Positive_Direction ; // Direction of movement mc_direction [ deafult mc_positive_direction]
	mcBuffermode: 	MC_BufferMode ; // Buffermode defines how the previous command is executed.
END_VAR
VAR
	xbNewCmdVelocity : BOOL ; // a new command velocity has been detected
END_VAR
// set blocked command if halt is active 
bBlockedCommand := fbMcHalt.Active ;

// Velocity conversion from RPM to deg/sec
	IF bIcfCmdVelocityRpm THEN 
		fVelocity := Rpm_To_DegS(fVelocity);
	END_IF

// check for command velocity changes
	IF fVelocity > 0 THEN 	
		xbNewCmdVelocity := fbMcMoveVelocity.Velocity <> fVelocity OR NOT fbMcMoveVelocity.Active ;
	ELSE
		bExec_Halt := TRUE;
		fbMcHalt.Deceleration	:= fCmdDecc;
		fbMcHalt.BufferMode		:= mcBuffermode	;
	END_IF
	
// Set command to true for one cycle
	IF (NOT AxisRef.Status.CmdBuffered OR mcBuffermode <> MC_Aborting) AND fVelocity > 0 THEN 
		bExec_MoveVelocityDynamic 	:= xbNewCmdVelocity;
		bInternalEnable				:= TRUE ;
	END_IF
	
// coppy parameters
	fbMcMoveVelocity.Velocity	:= fVelocity 	;
	fbMcMoveVelocity.Direction 	:= mcDirection	;
	fbMcMoveVelocity.BufferMode	:= mcBuffermode	;

// Set feedback output
	CmdMoveVelocityDynamic := fbMcMoveVelocity.Active ;
END_METHOD

METHOD PUBLIC CmdOverwriteAcc : BOOL // temporarilly overwrite deceleration values
VAR_INPUT	
	fValue	: LREAL ; // Overwrite value 
END_VAR
fAcceleration := fValue ;

CmdOverwriteAcc := TRUE ;
END_METHOD

METHOD PUBLIC CmdOverwriteDec : BOOL // Temporarilly overwrite deceleration values
VAR_INPUT
	fValue	: LREAL ; // Overwrite value 
END_VAR
fDeceleration := fValue ;

CmdOverwriteDec := TRUE ;
END_METHOD

METHOD PUBLIC CmdReset : BOOL
VAR_INPUT
END_VAR
// Set reset axis to true 				
	bExec_Reset 	:= TRUE ; 
	bInternalEnable	:= TRUE ;
	
// Set feedback output 
	CmdReset := tonResetDone.Q OR (AxisRef.Status.Coupled AND bResetDone) ;
END_METHOD

METHOD PUBLIC CmdSafeSpeed : BOOL
VAR_INPUT
END_VAR
// Set safestop command
bCmdSafeSpeed := TRUE ; 

// Set feedback output 
CmdSafeSpeed := fbMcPower.Override = fSafeOverride  ;
END_METHOD

METHOD PUBLIC CmdSafeStop : BOOL
VAR_INPUT
END_VAR
IF AxisRef.Status.Coupled THEN 
	CmdSafeStop := AxisRef.Status.NotMoving ;
	RETURN;
END_IF
// Set safestop command
bCmdSafeStop := TRUE ; 

// Set feedback output 
CmdSafeStop := bIsSafe OR NOT bInitOk;
END_METHOD

METHOD PUBLIC CmdSetPosition : BOOL
VAR_INPUT
	fPosition		: LREAL ; // encoder position
	bSetRelative	: BOOL 	; // TRUE = relative position offset, FALSE = Absolute position
END_VAR
bExec_SetPosition 			:= NOT fbMcSetPosition.Busy AND NOT fbMcSetPosition.Done ; 
fbMcSetPosition.Position	:= fPosition ;
fbMcSetPosition.Mode		:= bSetRelative ;

CmdSetPosition := fbMcSetPosition.Done;
END_METHOD

METHOD PRIVATE ExecEnable : BOOL
VAR_INPUT
END_VAR
// ===== Set axis enable ======
IF NOT bSafetyOk 
OR NOT bSTOOK 
OR AxisRef.Status.DriveDeviceError
OR bExec_Reset THEN 
	bCmdEnableAxis := FALSE ;
ELSIF bCmdManual AND bSafetyOk THEN 
	bCmdEnableAxis 	:= TRUE ;
	bInternalEnable S= bCmdManual ;
	bCmdManual 		:= FALSE ;
ELSE 
	bCmdEnableAxis	:= bEnable ;
END_IF

// ===== Check if axis is bussy with a command =====
	bInternalEnable S= AxisRef.Status.HasJob;
	bInternalEnable	S= bIcfAlwaysEnable ; // always enable axis if configured
	bInternalEnable	S= AxisRef.Status.Coupled ;

// ===== Axis disable timer after last command =====
	TofIntAxisEnable (	IN:= bInternalEnable, PT := tDisableDelay);

// ===== Enable drive =====
	fbMcPower(	Axis			:= AxisRef , 
				Enable			:= bCmdEnableAxis AND TofIntAxisEnable.Q, 
				Enable_Positive	:= bIcfEnableForward, 
				Enable_Negative	:= bIcfEnablereverse, 
				BufferMode		:= MC_Buffered );  
				
// ===== Reset internal enable signal =====
	bInternalEnable := FALSE ; 	

// ===== Delayed enable function =====	
	IF fbMcPower.Enable AND fbMcPower.Status THEN
		bAxisIsEnabled := TRUE ;
	ELSIF NOT fbMcPower.Enable OR AxisRef.Status.Error THEN 
		bAxisIsEnabled := FALSE ; 
	END_IF

	TonMotionEnable	(IN := bAxisIsEnabled, PT := tEnableDelay);
	bDelayedEnable 	:= TonMotionEnable.Q ;	

IF AxisRef.Status.DriveDeviceError 
AND bCmdEnableAxis THEN
	bError					:= TRUE							;
	stFault.Active 			:= TRUE 						;
	stFault.MessageNumber	:= E_MessageNumbers.FF_AxisFault;
	stFault.Discription		:= CONCAT('Drive device error ', UDINT_TO_STRING(AxisRef.Status.ErrorID));
	stFault.Discription		:= CONCAT( sName , stfault.Discription ) ;
	stFault.FaultType		:= E_FaultTypes.FF				;
ELSIF fbMcPower.Error THEN 
	bError					:= TRUE							;
	stFault.Active 			:= TRUE 						;
	stFault.MessageNumber	:= E_MessageNumbers.FF_AxisFault;
	stFault.Discription		:= CONCAT('Enable Fault ', UDINT_TO_STRING(fbMcPower.ErrorID));
	stFault.Discription		:= CONCAT( sName , stfault.Discription ) ;
	stFault.FaultType		:= E_FaultTypes.FF				;
END_IF
END_METHOD

METHOD INTERNAL ExecGearDynamic : BOOL
VAR_INPUT
END_VAR
// ===== invert gear ratio if reverse slave is active =====
	IF bReverseSlave THEN 
		fbMcGearInDyn.GearRatio := fCmdGearRatio * -1 ;
	ELSE 
		fbMcGearInDyn.GearRatio := fCmdGearRatio ;
	END_IF

// ===== Execute gear in function =====
	fbMcGearInDyn ( 	Master 			:= refMasterAxis,
						Slave			:= AxisRef,
						Enable 			:= bExec_GearSlaveDyn AND bDelayedEnable,
						Acceleration	:= 0,
						Deceleration	:= 0	); 
						
// ===== reset command =====
	bExec_GearSlaveDyn	:= FALSE ;
	bGearedAsSlave		:= fbMcGearInDyn.InGear ; 

// Gearing fault handling 
	IF fbMcGearInDyn.Error THEN 
		bError					:= TRUE							;
		stFault.Active 			:= TRUE 						;
		stFault.MessageNumber	:= E_MessageNumbers.FF_AxisFault;
		stFault.Discription		:= CONCAT('Gear dynamic Fault ', UDINT_TO_STRING(fbMcGearInDyn.ErrorID));	
		stFault.Discription		:= CONCAT( sName , stfault.Discription ) ;
		stFault.FaultType		:= E_FaultTypes.FF				;
	END_IF
END_METHOD

METHOD INTERNAL ExecGearIn : BOOL
VAR_INPUT
END_VAR
// ===== invert gear ratio if reverse slave is active =====
	IF bReverseSlave THEN 
		fbMcGearInSlave.RatioNumerator := fCmdGearRatio * -1 ;
	ELSE 
		fbMcGearInSlave.RatioNumerator := fCmdGearRatio ;
	END_IF

// ===== Execute gear in function =====
	fbMcGearInSlave ( 	Master 			:= refMasterAxis,
						Slave			:= AxisRef,
						Execute 		:= bExec_GearAsSlave AND bDelayedEnable,
						RatioDenominator:= 1,
						Acceleration	:= 0,
						Deceleration	:= 0	); 
						
// ===== reset command =====
	bExec_GearAsSlave 	:= FALSE  ;
	bGearedAsSlave		S= fbMcGearInSlave.InGear ; 

// Gearing fault handling 
	IF fbMcGearInSlave.Error THEN 
		bError					:= TRUE							;
		stFault.Active 			:= TRUE 						;
		stFault.MessageNumber	:= E_MessageNumbers.FF_AxisFault;
		stFault.Discription		:= CONCAT('Gear as slave Fault ', UDINT_TO_STRING(fbMcGearInSlave.ErrorID));
		stFault.Discription		:= CONCAT( sName , stfault.Discription ) ;
		stFault.FaultType		:= E_FaultTypes.FF				;
	END_IF
END_METHOD

METHOD INTERNAL ExecGearOut : BOOL
VAR_INPUT
END_VAR
// ===== execute gear out function ======
	fbMcGearOutSlave (	Slave 	:= AxisRef,
						Execute := bExec_GearOutSlave );

// ===== reset command =====
	bExec_GearOutSlave	:= false ;
	bGearedAsSlave		R= fbMcGearOutSlave.Done 	; 

// Gearing fault handling 
	IF fbMcGearOutSlave.Error THEN 
		bError					:= TRUE							;
		stFault.Active 			:= TRUE 						;
		stFault.MessageNumber	:= E_MessageNumbers.FF_AxisFault;
		stFault.Discription		:= CONCAT('Gear out Fault ', UDINT_TO_STRING(fbMcGearOutSlave.ErrorID));
		stFault.Discription		:= CONCAT( sName , stfault.Discription ) ;
		stFault.FaultType		:= E_FaultTypes.FF				;
	END_IF
END_METHOD

METHOD INTERNAL ExecHalt : BOOL
VAR_INPUT
END_VAR
// ==== Execute halt function ===== 
fbMcHalt (	Axis 		:= AxisRef,
			Execute 	:= bExec_Halt );

// ===== reset command =====
	bExec_Halt := FALSE ;
	
// Halt fault handling 
	IF fbMcHalt.Error THEN 
		bError					:= TRUE							;
		stFault.Active 			:= TRUE 						;
		stFault.MessageNumber	:= E_MessageNumbers.FF_AxisFault;
		stFault.Discription		:= CONCAT('Halt Fault ', UDINT_TO_STRING(fbMcHalt.ErrorID));
		stFault.Discription		:= CONCAT( sName , stfault.Discription ) ;
		stFault.FaultType		:= E_FaultTypes.FF				;
	END_IF
END_METHOD

METHOD INTERNAL ExecHome : BOOL
VAR_INPUT
END_VAR
// ==== execute homing function =====
	IF bIcfNCHomeSensor THEN 
		fbmchome.bCalibrationCam	:= NOT IAxisHome;
	ELSE
		fbmchome.bCalibrationCam	:= IAxisHome;
	END_IF		
		
	fbMcHome(	Axis			:= AxisRef,
				Execute			:= bExec_Home AND bDelayedEnable,
				HomingMode		:= mcHomingMode ); 
			
// Reset exec command 
	bExec_Home 	:= FALSE ;
	bHomed		S= fbMcHome.Done ;	
				
// fault handling 
	IF fbMcHome.Error THEN 
		bError					:= TRUE							;
		stFault.Active 			:= TRUE 						;
		stFault.MessageNumber	:= E_MessageNumbers.FF_AxisFault;
		stFault.Discription		:= CONCAT('Homing Fault ', UDINT_TO_STRING(fbMcHome.ErrorID));
		stFault.Discription		:= CONCAT( sName , stfault.Discription ) ;
		stFault.FaultType		:= E_FaultTypes.FF				;
	END_IF
END_METHOD

METHOD INTERNAL ExecJog : BOOL
VAR_INPUT
END_VAR
// ===== Execute Jog function =====
	IF bCmdLimitVelocity THEN 
		fbMcJog.Velocity := MIN(fCmdVelocityLimit, fbMcJog.Velocity); 
	END_IF

	// function call
	fbMcJog (	Axis 		:= AxisRef,
				JogForward	:= bExec_JogPositive AND bDelayedEnable,
				JogBackwards:= bExec_JogNegative AND bDelayedEnable,
				Acceleration:= fAcceleration,
				Deceleration:= fDeceleration );

// ===== reset command =====
	bExec_JogPositive 	:= FALSE  ;
	bExec_JogNegative	:= FALSE  ;
	
// Jog fault handling 
	IF fbMcJog.Error THEN 
		bError					:= TRUE							;
		stFault.Active 			:= TRUE 						;
		stFault.MessageNumber	:= E_MessageNumbers.FF_AxisFault;
		stFault.Discription		:= CONCAT('Jog Fault ', UDINT_TO_STRING(fbMcJog.ErrorID));
		stFault.Discription		:= CONCAT( sName , stfault.Discription ) ;
		stFault.FaultType		:= E_FaultTypes.FF				;
	END_IF
END_METHOD

METHOD INTERNAL ExecMoveAbsolute : BOOL
VAR_INPUT
END_VAR
// ==== execute move absolute function =====
FOR i := 0 TO 1 DO 
	// Limit velocity
	IF bCmdLimitVelocity THEN 
		fbMcJog.Velocity := MIN(fCmdVelocityLimit, fbMcMoveAbsolute[i].Velocity); 
	END_IF
	// function call
	fbMcMoveAbsolute[i](	Axis 		:= AxisRef,
							Execute 	:= arExec_MoveAbs[i] AND bDelayedEnable,
							Acceleration:= fAcceleration,
							Deceleration:= fDeceleration );  

	// If function is done then reset command values
	IF fbMcMoveAbsolute[i].Done OR fbMcMoveAbsolute[i].CommandAborted OR NOT arExec_MoveAbs[i] THEN 
		fbMcMoveAbsolute[i].Velocity	:= 0 ;
		fbMcMoveAbsolute[i].Position	:= 0 ; 
	END_IF

	// reset Exec command 
	arExec_MoveAbs[i] := FALSE ; 
	
	// fault handling 
	IF fbMcMoveAbsolute[i].Error THEN 
		bError					:= TRUE							;
		stFault.Active 			:= TRUE 						;
		stFault.MessageNumber	:= E_MessageNumbers.FF_AxisFault;
		stFault.Discription		:= CONCAT('Move absolute Fault ', UDINT_TO_STRING(fbMcMoveAbsolute[i].ErrorID));
		stFault.Discription		:= CONCAT( sName , stfault.Discription ) ;
		stFault.FaultType		:= E_FaultTypes.FF				;
	END_IF
END_FOR
END_METHOD

METHOD INTERNAL ExecMoveModulo : BOOL
VAR_INPUT
END_VAR


// ===== Execute move modulo function =====
FOR i := 0 TO 1 DO 
	IF bCmdLimitVelocity THEN 
		fbMcJog.Velocity := MIN(fCmdVelocityLimit, fbMcMoveModulo[i].Velocity); 
	END_IF
	// function call
	fbMcMoveModulo[i](	Axis 		:= AxisRef,
						Execute 	:= arExec_MoveModulo[i] AND bDelayedEnable,
						Acceleration:= fAcceleration,
						Deceleration:= fDeceleration);  
	
	// If function is done then reset command values
	IF fbMcMoveModulo[i].Done OR fbMcMoveModulo[i].CommandAborted OR NOT arExec_MoveModulo[i] THEN 
		fbMcMoveModulo[i].Velocity	:= 0 ;
		fbMcMoveModulo[i].Position	:= 0 ; 
	END_IF

	// reset Exec command 
	arExec_MoveModulo[i] := FALSE ; 
	
	// fault handling 
	IF fbMcMoveModulo[i].Error THEN 
		bError					:= TRUE							;
		stFault.Active 			:= TRUE 						;
		stFault.MessageNumber	:= E_MessageNumbers.FF_AxisFault;
		stFault.Discription		:= CONCAT('Move module Fault ', UDINT_TO_STRING(fbMcMoveModulo[i].ErrorID));
		stFault.Discription		:= CONCAT( sName , stfault.Discription ) ;
		stFault.FaultType		:= E_FaultTypes.FF			;
	END_IF
END_FOR
END_METHOD

METHOD INTERNAL ExecMoveRelative : BOOL
VAR_INPUT
END_VAR
//ReCmd_MoveModulo(CLK := bCmd_MoveModulo );
//bCmd_MoveModulo	:= FALSE ;

// ===== Execute move relative function ======
FOR i := 0 TO 1 DO 
	// Limit velocity
	IF bCmdLimitVelocity THEN 
		fbMcJog.Velocity := MIN(fCmdVelocityLimit, fbMcMoveModulo[i].Velocity); 
	END_IF
	// function call
	fbMCMoveRelative[i](	Axis 		:= AxisRef,
							Execute		:= arExec_MoveRelative[i] AND bDelayedEnable,
							Acceleration:= fAcceleration,
							Deceleration:= fDeceleration );

	// If function is done then reset command values
	IF fbMCMoveRelative[i].Done OR fbMCMoveRelative[i].CommandAborted OR NOT arExec_MoveRelative[i] THEN 
		fbMCMoveRelative[i].Velocity	:= 0 ;
		fbMCMoveRelative[i].Distance	:= 0 ; 
	END_IF

	// reset Exec command 
	arExec_MoveRelative[i] := FALSE ; 
	
	// fault handling 
	IF fbMCMoveRelative[i].Error THEN 
		bError					:= TRUE							;
		stFault.Active 			:= TRUE 						;
		stFault.MessageNumber	:= E_MessageNumbers.FF_AxisFault;
		stFault.Discription		:= CONCAT('Move relative Fault ', UDINT_TO_STRING(fbMCMoveRelative[i].ErrorID));
		stFault.Discription		:= CONCAT( sName , stfault.Discription ) ;
		stFault.FaultType		:= E_FaultTypes.FF			;
	END_IF
END_FOR
END_METHOD

METHOD INTERNAL ExecMoveVelocity : BOOL
VAR_INPUT
END_VAR
// ===== Execute move velocity function =====
	IF bCmdLimitVelocity THEN 
		fbMcJog.Velocity := MIN(fCmdVelocityLimit, fbMcMoveVelocity.Velocity); 
	END_IF

// function call
fbMcMoveVelocity (	Axis 		:= AxisRef,
					Execute		:= (bExec_MoveVelocity OR bExec_MoveVelocityDynamic) AND bDelayedEnable,
					Acceleration:= fAcceleration,
					Deceleration:= fDeceleration );

// ===== reset command =====
bExec_MoveVelocity 			:= FALSE ;
bExec_MoveVelocityDynamic 	:= FALSE;
	
// Halt fault handling 
IF fbMcMoveVelocity.Error THEN 
	bError					:= TRUE							;
	stFault.Active 			:= TRUE 						;
	stFault.MessageNumber	:= E_MessageNumbers.FF_AxisFault;
	stFault.Discription		:= CONCAT('Move velocity Fault ', UDINT_TO_STRING(fbMcMoveVelocity.ErrorID));
	stFault.Discription		:= CONCAT( sName , stfault.Discription ) ;
	stFault.FaultType		:= E_FaultTypes.FF				;
END_IF
END_METHOD

METHOD INTERNAL ExecReadStatus : BOOL
VAR_INPUT
END_VAR
AxisRef.ReadStatus();
					
// convert velocity to RPM for output if aplicable
IF bIcfCmdVelocityRpm THEN 
	fVelocity := AxisRef.NcToPlc.ActVelo / 6 ;
ELSE 
	fVelocity := AxisRef.NcToPlc.ActVelo ;
END_IF

// write position output
IF bIcfModuloAxis THEN 
	fActPosition := AxisRef.NcToPlc.ModuloActPos ;
ELSE
	fActPosition := AxisRef.NcToPlc.ActPos ;
END_IF
						
// set status bits 
bIdle := NOT AxisRef.Status.HasJob ;

// In position 
	rtrigInPosition( 	CLK := AxisRef.Status.InTargetPosition, 
						Q => bReInTargetPos);
END_METHOD

METHOD INTERNAL ExecReset : BOOL
VAR_INPUT
END_VAR
VAR
	xMcReset			: BOOL ; // Execute MC reset
	xSoeReset			: BOOL ; // Execute SOE reset

END_VAR
//IF  AxisRef.Status.Moving AND bExec_Reset THEN // If the axis is still moving execute safe stop first
//	RETURN;
IF AxisRef.Status.Coupled THEN 
	bResetDone 	:= NOT AxisRef.Status.Error;
	bExec_Reset	R= bResetDone  ;
	RETURN;
END_IF

// ===== reset command =====
	bError 		:= AxisRef.Status.Error ; 
	bExec_Reset	R= fbMcReset.Done  ;

// ==== execute reset functions =====
IF AxisRef.Status.DriveDeviceError AND IAxisSTOOK THEN 
		xSoeReset := TRUE ;
ELSIF bSTOOK AND bExec_Reset THEN
		xMcReset	:= TRUE ;
ELSE 
	xSoeReset 	:= FALSE ;
	xMcReset	:= FALSE ;
END_IF

fbSoeReset	( 	Execute := xSoeReset,
				Timeout	:= T#5S,
				Axis	:= AxisRef);

fbMcReset	( 	Execute	:= xMcReset,
				Axis	:= AxisRef ); 
				
// ===== Set feedback =====
	bResetDone 	S= fbMcReset.Done  ;
	bResetDone	R= AxisRef.Status.Error ;
	tonResetDone (IN	:= bResetDone);

// ===== reset limitations =====
	bCmdSafeSpeed 	:= FALSE ;

	
// Reset fault handling 
	IF fbSoeReset.Error OR fbMcReset.Error THEN 
		bError					:= TRUE							;
		stFault.Active 			:= TRUE 						;
		stFault.MessageNumber	:= E_MessageNumbers.FF_AxisFault;
		stFault.Discription		:= CONCAT('Reset Fault ', UDINT_TO_STRING(fbMcReset.ErrorID));
		stFault.Discription		:= CONCAT( sName , stfault.Discription ) ;
		stFault.FaultType		:= E_FaultTypes.FF				;
	END_IF
END_METHOD

METHOD PRIVATE ExecSafeFunctions : BOOL
VAR_INPUT
END_VAR
// ==== Stop when safety is not ok =====
	bCmdSafeStop S= NOT bSafetyOk ;

// ===== Safe torque off function =====
	IF bIcfSTOPresent THEN 
		tonSTOOK(IN := IAxisSTOOK, PT := T#1000MS);
		bSTOOK := tonSTOOK.Q AND NOT AxisRef.Status.DriveDeviceError;
//		bSTOOK	:= IAxisSTOOK ;
	ELSE 
		bSTOOK := true ;
	END_IF
	
// ==== Safe operation functions (overrule all other motion functions) =====
	IF NOT AxisRef.Status.Coupled AND bSTOOK THEN 
		fbMcStop( 	Axis 			:= AxisRef		,
					Execute 		:= bCmdSafeStop AND NOT bExec_Reset,
					Deceleration	:= fMaxDec		);
	END_IF
	
	// Reset axis command			
	bCmdSafeStop 	R= fbMcStop.Done OR AxisRef.Status.HasBeenStopped OR NOT bSTOOK ;
	bStopped		:= AxisRef.Status.HasBeenStopped OR NOT bSTOOK ;

// Safestop fault handling 
	IF fbMcStop.Error THEN 
		bError					:= TRUE							;
		stFault.Active 			:= TRUE 						;
		stFault.MessageNumber	:= E_MessageNumbers.FF_AxisFault;
		stFault.Discription		:= CONCAT('Safe stop axis fault ', UDINT_TO_STRING(fbMcStop.ErrorID));
		stFault.Discription		:= CONCAT( sName , stfault.Discription ) ;
		stFault.FaultType		:= E_FaultTypes.FF				;
	END_IF
	
// ===== Safe speed monitoring =====
	IF bCmdSafeSpeed THEN 
		fbMcPower.Override 	:= fSafeOverride ;
		bCmdSafeSpeed		:= FALSE ;
	ELSE 
		fbMcPower.Override := 100 ;
	END_IF

// ===== Dev is safe feedback =====
bIsSafe := AxisRef.Status.HasBeenStopped OR AxisRef.Status.Disabled  ;
END_METHOD

METHOD INTERNAL ExecSetPosition : BOOL
VAR_INPUT
END_VAR
// ====== set position of axis ======
IF bExec_SetPosition OR fbMcSetPosition.Busy THEN 
	fbMcSetPosition (	Axis 	:= AxisRef,
						Execute	:= bExec_SetPosition );
	bExec_SetPosition := TRUE ;
END_IF
END_METHOD

METHOD PRIVATE ExecWriteParameter : BOOL
VAR_INPUT
END_VAR
// check if axis is disabled before writeing parameter
	AxisRef.ReadStatus();
	IF AxisRef.Status.Disabled 
	AND (fbMcWriteParameter.Busy OR bExec_ParWritePers) THEN
		fbMcWriteParameter	( 	Axis 	:= AxisRef,
								Execute	:= bExec_ParWritePers );
	ELSE
		fbMcWriteParameter.Execute := FALSE ; 
		RETURN;
	END_IF
						
// fault handling 
	IF fbMcWriteParameter.Error THEN 
		bError					:= TRUE							;
		stFault.Active 			:= TRUE 						;
		stFault.MessageNumber	:= E_MessageNumbers.FF_AxisFault;
		stFault.Discription		:= CONCAT('Cannot write parameter Id#:', UDINT_TO_STRING(fbMcHome.ErrorID));
		stFault.Discription		:= CONCAT( sName , stfault.Discription ) ;
		stFault.FaultType		:= E_FaultTypes.FF				;
	END_IF
 
// reset commands
	bExec_ParWritePers := FALSE ;
END_METHOD

METHOD PUBLIC Init : BOOL
VAR_INPUT
	// Message location data
	nId			: UDINT ; // Identification number of object
	nParentId	: UDINT ; // Id of higher level If aplicable (0 = no parent)
	// Config Bits
	bIcfCmdVelocityRpm	: BOOL := FALSE ; // input speeds in Rpm
	bIcfEnableForward 	: BOOL := TRUE 	; // Enable forward motion
	bIcfEnablereverse	: BOOL := TRUE 	; // Enable reverse motion
	bIcfAlwaysEnable	: BOOL := FALSE ; // 1 = Axis always enabled, 0 = Axis disabled at Idle 
	bIcfSimulationMode	: BOOL := FALSE ; // Simulation mode is active [default set to False] Used for testing without hardware present 
	bIcfModuloAxis		: BOOL := FALSE ; // Show axis position as modulo
	bIcfSTOPresent		: BOOL := FALSE ; // Axis safe torque off is present
	bIcfNCHomeSensor	: BOOL := FALSE ; // Homing sensor is inverted (NC)	
	// Config Values 
	mcHomingMode 		: MC_HomingMode := MC_HomingMode.MC_DefaultHoming; 
	fHomePosition		: LREAL := 0 	; // set position at homing
	fSafeOverride		: LREAL := 10	; // Safe velocity override [%]
	nEncTurnoverVal 	: LREAL := 360	; // encoder turnover value 
	tEnableDelay		: time 	:= T#0MS; // Time between axis enable command and motion command execution (0 := no delay active)	
	tDisabledelay		: TIME 	:= T#100MS; // Axis idle time before axis is disabled 
END_VAR
VAR 
	bActVeloReadValid 	: BOOL ; // velocity parameter read is valid 
	bActAccReadValid 	: BOOL ; // Acceleration parameter read is valid 
	bActDecReadValid 	: BOOL ; // Deceleration parameter read is valid 
	bActParamValid 		: BOOL ; // Parameter read is valid 
END_VAR
// ====== Set init to true =====
	bInitOk	:= TRUE ; 

// ====== Calculate device id =====
	bInitOk :=	ExecIdentifyDevice(nId,nParentId, E_ComponentTypes.Axis) AND bInitOk;

// ====== Set manual device type ======
	eDevType := E_Devices.Axis ;	
	
// ===== Message data set =====
	stFault.ComponentType		:= E_ComponentTypes.Axis ;
	
// ===== Read system configuration =====
	McReadSysVelo	(	Axis 			:= AxisRef,
						Enable 			:= Cmd_EnDriveParRead ,
						ParameterNumber := MaxVelocitySystem ,
						ReadMode		:= 1,
						Valid			=> bActVeloReadValid ,						
						Busy			=> ,
						Error			=> ,
						ErrorID			=> ,
						Value			=> fMaxVelo );
	McReadSysAcc	(	Axis 			:= AxisRef,
						Enable 			:= Cmd_EnDriveParRead ,
						ParameterNumber := MaxAccelerationSystem ,
						ReadMode		:= 1,
						Valid			=> bActAccReadValid ,						
						Busy			=> ,
						Error			=> ,
						ErrorID			=> ,
						Value			=> fMaxAcc );
	McReadSysDec	(	Axis 			:= AxisRef,
						Enable 			:= Cmd_EnDriveParRead ,
						ParameterNumber := MaxDecelerationSystem ,
						ReadMode		:= 1,
						Valid			=> bActDecReadValid ,						
						Busy			=> ,
						Error			=> ,
						ErrorID			=> ,
						Value			=> fMaxDec );

	IF 	fMaxVelo > 0 
	AND fMaxAcc >0
	AND fMaxDec >0 THEN 
		bActParamValid	:= TRUE ; 
		fCmdAcc 		:= fMaxAcc * 0.9;
		fCmdDecc		:= fMaxDec * 0.9;
	END_IF

	IF NOT Cmd_EnDriveParRead AND NOT bActParamValid THEN  
		Cmd_EnDriveParRead := TRUE;
	ELSIF Cmd_EnDriveParRead THEN
		Cmd_EnDriveParRead := FALSE;
	END_IF

// ===== Configure Axis =====
	// ***** Config Bits *****
		THIS^.bIcfCmdVelocityRpm	:= bIcfCmdVelocityRpm	; // Enable speed inputs in Rpm
		THIS^.bIcfEnableForward 	:= bIcfEnableForward 	; // Enable forward motion
		THIS^.bIcfEnablereverse		:= bIcfEnablereverse	; // Enable reverse motion
		THIS^.bIcfAlwaysEnable		:= bIcfAlwaysEnable		; // Always enable motor and brake if safety is ok
		THIS^.bIcfSimulationMode	:= bIcfSimulationMode 	; // Simulation mode is active [default set to False] 
		THIS^.bIcfModuloAxis		:= bIcfModuloAxis		; // show axis position as modulo
		THIS^.bIcfSTOPresent		:= bIcfSTOPresent		; // Axis has safe torque off function
		THIS^.bIcfNCHomeSensor		:= bIcfNCHomeSensor		; // Axis homing sensor is NC	
	// ***** config homing Mode ***** 
 		THIS^.mcHomingMode 			:= mcHomingMode ; // set homing mode
		THIS^.fHomePosition			:= fHomePosition;
	// ***** Velocity settings *****
		THIS^.fSafeOverride			:= fSafeOverride	; 	
	// ***** Encoder values *****
		THIS^.fEncoderTurnoverValue := nEncTurnoverVal	; // turnover value for encoder = 25.6 mm per rev * 4096 revolutions 
	// ***** Time delay enable off *****
		THIS^.tEnableDelay		:= tEnableDelay	;
		THIS^.tDisableDelay 	:= tDisabledelay ;		
		
// ===== configure parameters =====
	ParAccManualScaling.fMinimum 		:= 1 	;
	ParAccManualScaling.fMaximum		:= 100 	;
	ParAccManualScaling.nNumber 		:= nLocationId + 1;
	ParAccManualScaling.sDiscription  	:= CONCAT( STR1 := sName, STR2 := 'percantage of acceleration used For jogging');
	ParAccManualScaling.sName			:= CONCAT( STR1 := sName, STR2 := 'Manual acc scaling');
	ParAccManualScaling.sType			:= 'Mpar';
	ParAccManualScaling.sUnit			:= '%';
	refFbParHandler.CmdAddParameter( refParameter := ParAccManualScaling );

	
	ParDecManualScaling.fMinimum 		:= 1 	;
	ParDecManualScaling.fMaximum		:= 100 	;
	ParDecManualScaling.nNumber 		:= nLocationId + 2;
	ParDecManualScaling.sDiscription  	:= CONCAT( STR1 := sName, STR2 := 'percantage of deceleration used For jogging');
	ParDecManualScaling.sName			:= CONCAT( STR1 := sName, STR2 := 'Manual dec scaling');
	ParDecManualScaling.sType			:= 'Mpar';
	ParDecManualScaling.sUnit			:= '%';
	refFbParHandler.CmdAddParameter( refParameter := ParAccManualScaling );

// ===== reset axis state indicators ======
	bError 	:= FALSE;

// ====== Set init to done =======
bInitOk := bActParamValid AND bInitOk;
Init := bInitOk;
END_METHOD

END_FUNCTION_BLOCK

// ---- Heaters/FB_DevDoublePWM.TcPOU
{attribute 'reflection'}
FUNCTION_BLOCK PUBLIC FB_DevDoublePWM EXTENDS FB_DevBase // PWM control for 2 outputs that cannot be switchid on simultaniously
VAR_INPUT
	bCmdPWMOn			: BOOL := FALSE ; // PWM controller on 
END_VAR
VAR_OUTPUT
END_VAR
VAR
	bCmdChanelAOn		: BOOL := FALSE ; // command switch chanel A on permanently
	bCmdChanelBOn		: BOOL := FALSE ; // Commandswitch chanel B on permanently 
	bCmdOverrulePWM		: BOOL := FALSE ; // Command to overrule PWM
	bCmdHold			: BOOL := false ; // Command hold PWM on signals (collision avoidance)

	tPeriodLength		: TIME  ; // desired PWM cycle time length [ms] 
	tDutyCycle 			: TIME	; // percentage of power [%]
	tIdleTime			: TIME	; // Time both outputs are idle during PWM
	
	tonOutputA 			: TON ; // Timer on PWM output A
	tonOutputB 			: TON ; // Timer on PWM output B
	tonIdle				: TON ; // Timer On PWM Idle time (both outputs off)

	tofOutputA 			: TOF ; // Timer off PWM output A Off (For overlap prevention)
	tofOutputB 			: TOF ; // Timer off PWM output B Off ( for overlap prevention)

	stParPeriodLength	: Udt_Parameter := (fValue := 2000); // desired PWM cycle time length [ms] Parameter
	stParDutyCycle 		: Udt_Parameter	:= ( fValue := 0); // percentage of power [%] Parameter
	stParSwitchOverTime	: Udt_Parameter	; // Time between switching A off and B on (and vice versa) Parameter
	stMaxTimeOn			: Udt_Parameter := (fValue := 1000);// Maximum time a heater can be on without burning through
	
	qbOutputMain AT %Q* 	: BOOL 	; // physical output to main relais
	qbOutputA	 AT %Q* 	: BOOL 	; // physical output to output A
	qbOutputB	 AT %Q* 	: BOOL 	; // physical output to output B
	
	nPWMStep	: INT ; // PWM stepper

	tonBurnTimeA	: TON ; // burn timer for coil A
	tonBurnTimeB	: TON ; // burn timer for coil B 
END_VAR

// set device type
IF eDevType = E_Devices.Undefined THEN 
	eDevType := E_Devices.DoublePWMController ;
END_IF

// Call base function
SUPER^(refFbFault := refFbFault);


// ===== hold all actions if not initialized ======
IF NOT bInitOk THEN
	RETURN;
END_IF 

// call Functions 
CalcCycleTimes();
IF tDutyCycle > T#0S AND tPeriodLength > T#0S THEN // switch PWM controller up when cycle timer is null
	ExecPWMCycle(); // 
END_IF 

ExecSetOutputs();

METHOD INTERNAL CalcCycleTimes : BOOL // calculate cycle timers
VAR_INPUT
END_VAR
VAR 
END_VAR
// Calculate Cycle timers
tPeriodLength	:= LREAL_TO_TIME( stParPeriodLength.fValue );
tDutyCycle		:= LREAL_TO_TIME(stParPeriodLength.fValue * (stParDutyCycle.fValue / 100));
tIdleTime		:= LREAL_TO_TIME(stParPeriodLength.fValue) - (tDutyCycle * 2) ;

tofOutputA.PT := LREAL_TO_TIME(stParSwitchOverTime.fValue);
tofOutputB.PT := LREAL_TO_TIME(stParSwitchOverTime.fValue);
END_METHOD

METHOD PUBLIC CmdHold : BOOL
VAR_INPUT
END_VAR
bCmdHold := TRUE ;

CmdHold := NOT qbOutputMain ;
END_METHOD

METHOD PUBLIC CmdOutputAOn : BOOL // Turn on chanel A permanently 
VAR_INPUT
END_VAR
bCmdOverrulePWM S= TRUE ;
bCmdChanelAOn S= TRUE ;

CmdOutputAOn := qbOutputA AND qbOutputMain ;
END_METHOD

METHOD PUBLIC CmdOutputBOn : BOOL
VAR_INPUT
END_VAR
bCmdOverrulePWM S= TRUE ;
bCmdChanelBOn S= TRUE ;

CmdOutputBOn := qbOutputB AND qbOutputMain ;
END_METHOD

METHOD PUBLIC CmdSafeStop : BOOL
VAR_INPUT
END_VAR
bCmdOverrulePWM S= TRUE ;
bCmdChanelAOn 		:= FALSE ;
bCmdChanelBOn		:= FALSE ;
qbOutputMain 		:= FALSE ;

bIsSafe := NOT (qbOutputA OR qbOutputB OR qbOutputMain);
END_METHOD

METHOD INTERNAL ExecPWMCycle : BOOL
VAR_INPUT
END_VAR
IF bCmdPWMOn THEN 
	IF bCmdOverrulePWM OR bCmdHold THEN 
		IF bCmdChanelAOn THEN 
			nPWMStep := 1 ;
		ELSE 
			nPWMStep := 0 ;
		END_IF
		bCmdOverrulePWM := FALSE ;
		RETURN;
	END_IF
ELSE 
	RETURN;
END_IF

// PWM stepper 
CASE nPWMStep OF 
	0: // Switch on chanel A
		bCmdChanelAOn := TRUE ;
		IF tonOutputA.Q THEN
			nPWMStep := 1 ;
		END_IF
	1: // Switch on chanel B
		bCmdChanelBOn := TRUE;
		IF tonOutputB.Q THEN
			nPWMStep := 2 ;
		END_IF
	2: // Idle Time 
		IF tonIdle.Q THEN 
			nPWMStep := 0;
		END_IF
	ELSE
		;
END_CASE

// call timers 
tonOutputA	(IN := bCmdChanelAOn, PT := tDutyCycle);
tonOutputB	(IN := bCmdChanelBOn, PT := tDutyCycle);
tonIdle 	(IN := nPWMStep = 2	, PT := tIdleTime);
END_METHOD

METHOD PRIVATE ExecSetOutputs : BOOL
VAR_INPUT
END_VAR

// Set main output
qbOutputMain := (bEnable OR bManual) AND bSafetyOk AND NOT bCmdHold ;

// Set outputs
qbOutputA := bCmdChanelAOn AND NOT tofOutputB.Q AND NOT tonBurnTimeA.Q;
qbOutputB := bCmdChanelBOn AND NOT tofOutputA.Q AND NOT tonBurnTimeB.Q;

// Call timers for overlap prevention
tofOutputA(IN := qbOutputA);
tofOutputB(IN := qbOutputB);

// reset commands
bCmdChanelAOn := FALSE ;
bCmdChanelBOn := FALSE ;

tonBurnTimeA ( IN := bCmdChanelAOn, PT := LREAL_TO_TIME( stMaxTimeOn.fValue));
tonBurnTimeB ( IN := bCmdChanelBOn, PT := LREAL_TO_TIME( stMaxTimeOn.fValue));

IF tonBurnTimeA.Q THEN 
	stFault.Active 			:= TRUE ;
	stFault.Discription 	:= 'Heater A burn timeout';
	stFault.MessageNumber 	:= E_MessageNumbers.CF_MoveToSlow ;
	stFault.FaultType		:= E_FaultTypes.CF;
	qbOutputA 				:= FALSE ;
ELSIF tonBurnTimeB.Q THEN 
	stFault.Active 			:= TRUE ;
	stFault.Discription 	:= 'Heater B burn timeout';
	stFault.MessageNumber 	:= E_MessageNumbers.CF_MoveToSlow ;
	stFault.FaultType		:= E_FaultTypes.CF;
	qbOutputB 				:= FALSE ;
END_IF

bCmdHold := FALSE ;
END_METHOD

METHOD PUBLIC Init : BOOL
VAR_INPUT
	// Message location data
	nId			: UDINT ; // Identification number of object
	nParentId	: UDINT ; // Id of higher level If aplicable (0 = no parent)
END_VAR
// ====== Set init to true =====
	bInitOk	:= TRUE ; 

// ====== Calculate device id =====
	bInitOk :=	ExecIdentifyDevice(nId,nParentId, E_ComponentTypes.Heaters) AND bInitOk;

// ====== Set message information =======
	stFault.ComponentType	:= E_ComponentTypes.Heaters	;

// ======= Reset Error bit ======
	bErrorActive 	:= FALSE;
	bBussy			:= FALSE;
	
// ===== configure parameters =====
	stParPeriodLength.fMinimum 		:= 0 		;
	stParPeriodLength.fMaximum		:= 60000 	;
	stParPeriodLength.nNumber 		:= nLocationId + 1;
	stParPeriodLength.sDiscription  := CONCAT( STR1 := sName, STR2 := 'Period length of the cycle in miliseconds');
	stParPeriodLength.sName			:= CONCAT( STR1 := sName, STR2 := 'Period Length');
	stParPeriodLength.sType			:= 'MPar';
	stParPeriodLength.sUnit			:= 'ms';
	stParPeriodLength.fValue		:= 5000;

	stParDutyCycle.fMinimum 		:= 0 		;
	stParDutyCycle.fMaximum			:= 50 		;
	stParDutyCycle.nNumber 			:= nLocationId + 2;
	stParDutyCycle.sDiscription  	:= CONCAT( STR1 := sName, STR2 := 'Percentage of period length in which an output is active');
	stParDutyCycle.sName			:= CONCAT( STR1 := sName, STR2 := 'Duty Cyle');
	stParDutyCycle.sType			:= 'MPar';
	stParDutyCycle.sUnit			:= '%';
	stParPeriodLength.fValue		:= 10;

	
	stParSwitchOverTime.fMinimum 	:= 0 		;
	stParSwitchOverTime.fMaximum	:= 500 		;
	stParSwitchOverTime.nNumber 	:= nLocationId + 3;
	stParSwitchOverTime.sDiscription:= CONCAT( STR1 := sName, STR2 := 'Idle time between output chanel switchover in miliseconds');
	stParSwitchOverTime.sName		:= CONCAT( STR1 := sName, STR2 := 'Switch Time');
	stParSwitchOverTime.sType		:= 'CPar';
	stParSwitchOverTime.sUnit		:= 'ms';

	stMaxTimeOn.fMinimum 	:= 0 		;
	stMaxTimeOn.fMaximum	:= 5000 	;
	stMaxTimeOn.nNumber 	:= nLocationId + 4;
	stMaxTimeOn.sDiscription:= CONCAT( STR1 := sName, STR2 := 'Maximum time a heater can be fully on without burning through');
	stMaxTimeOn.sName		:= CONCAT( STR1 := sName, STR2 := 'Max heating time');
	stMaxTimeOn.sType		:= 'MPar';
	stMaxTimeOn.sUnit		:= 'ms';
	
	
	// add parameters to handler 
	refFbParHandler.CmdAddParameter( refParameter := stParPeriodLength );
	refFbParHandler.CmdAddParameter( refParameter := stParDutyCycle );
	refFbParHandler.CmdAddParameter( refParameter := stParSwitchOverTime );
END_METHOD

END_FUNCTION_BLOCK

// ---- Sensors/AnalogInput/FunctionBlocks/FB_DevAnalogInputScaled.TcPOU
{attribute 'reflection'}
FUNCTION_BLOCK PUBLIC FB_DevAnalogInputScaled EXTENDS FB_DevAnalogInput
VAR_INPUT
END_VAR
VAR_OUTPUT
END_VAR
VAR
	nLimitMin		: INT := Utilities_Library.GVL_FixedValues.nINTMINVALUE	; // Initial value is set to integer minimum value for use with normal def analog inputs 
	nLimitMax 		: INT := Utilities_Library.GVL_FixedValues.nINTMAXVALUE	; // Initial value is set to integer minimum value for use with high def analog inputs
	fGainFactor 	: LREAL	:= 1	;
	nOfset			: INT	:= 0	;
END_VAR

SUPER^(refFbFault := refFbFault);

METHOD ExecSetFeedback : BOOL
VAR
	nCalibValue	: INT ; 
END_VAR
// Offset 
IF bCmdSimulate THEN 
	nCalibValue := fSimValue + nOfset ;
ELSE
	nCalibValue := inHwInput + nOfset ;
END_IF

fValue := INT_TO_LREAL(nCalibValue) / fGainFactor;

ExecSetFeedback := TRUE;
END_METHOD

METHOD PUBLIC SetScaling : BOOL 
VAR_INPUT
	fMaxValue	: LREAL ; 	// Maximum input value after scaling, e.g. 100%, 0 = no scaling (gain = hardware limit / fMaxValue)  
	fOfset		: LREAL ;	// offset value (fvalue = (gain * hwvalue) + fOfset)
END_VAR
// calculate gain 
IF fMaxValue =0 THEN 
	fGainFactor := 1 ;
ELSE 
	fGainFactor := nLimitMax / fMaxValue ;
END_IF

nOfset := LREAL_TO_INT(fOfset * fGainFactor) ;

SetScaling := TRUE;
END_METHOD

END_FUNCTION_BLOCK
